  MoveL 2523 to (502.47, 492.57, 5) mm, rotated rx 0 ry 90 rz 0 deg; joints [-11.281, -26.8, 110.891, -15.281, -83.436, 50.783]
  Set speed (30.0 mm/s)
  Call Extruder(0.229)
  MoveL 2524 to (508.03, 498.13, 5) mm, rotated rx 0 ry 90 rz 0 deg; joints [-11.685, -26.677, 110.09, -15.709, -82.794, 51.008]
  MoveL 2525 to (508.16, 498.26, 5) mm, rotated rx 0 ry 90 rz 0 deg; joints [-11.694, -26.674, 110.072, -15.719, -82.78, 51.013]
  Set speed (120.0 mm/s)
  MoveL 2526 to (509.32, 490.68, 5) mm, rotated rx 0 ry 90 rz 0 deg; joints [-10.985, -26.681, 110.115, -15.004, -82.793, 50.925]
  Set speed (30.0 mm/s)
  Call Extruder(0.767)
  MoveL 2527 to (490.68, 509.32, 5) mm, rotated rx 0 ry 90 rz 0 deg; joints [-13.056, -26.94, 111.861, -17.04, -84.281, 50.715]
  MoveL 2528 to (490.56, 509.44, 5) mm, rotated rx 0 ry 90 rz 0 deg; joints [-13.07, -26.942, 111.873, -17.054, -84.29, 50.713]
  Set speed (120.0 mm/s)
  MoveL 2529 to (501.29, 492.36, 5) mm, rotated rx 0 ry 90 rz 0 deg; joints [-11.283, -26.822, 111.037, -15.28, -83.556, 50.75]
  Set speed (1000.0 mm/s)
  MoveL 2530 to (501.36, 492.29, 5) mm, rotated rx 0 ry 90 rz 0 deg; joints [-11.276, -26.821, 111.031, -15.272, -83.55, 50.751]
  Set speed (15.0 mm/s)
  Call Extruder(0.010)
  MoveL 2531 to (501.71, 492.29, 5) mm, rotated rx 0 ry 90 rz 0 deg; joints [-11.269, -26.815, 110.989, -15.267, -83.516, 50.76]
  Call Extruder(0.064)
  MoveL 2532 to (503.91, 492.29, 5) mm, rotated rx 0 ry 90 rz 0 deg; joints [-11.229, -26.775, 110.726, -15.233, -83.299, 50.815]
  Call Extruder(0.055)
  MoveL 2533 to (503.91, 490.4, 5) mm, rotated rx 0 ry 90 rz 0 deg; joints [-11.056, -26.782, 110.77, -15.057, -83.331, 50.787]
  Call Extruder(0.166)
  MoveL 2534 to (509.6, 490.4, 5) mm, rotated rx 0 ry 90 rz 0 deg; joints [-10.955, -26.677, 110.087, -14.974, -82.77, 50.927]
  Call Extruder(0.233)
  MoveL 2535 to (509.6, 498.42, 5) mm, rotated rx 0 ry 90 rz 0 deg; joints [-11.681, -26.646, 109.894, -15.711, -82.636, 51.053]
  Call Extruder(0.057)
  MoveL 2536 to (507.66, 498.42, 5) mm, rotated rx 0 ry 90 rz 0 deg; joints [-11.718, -26.683, 110.128, -15.741, -82.826, 51.003]
  Call Extruder(0.072)
  MoveL 2537 to (507.66, 500.9, 5) mm, rotated rx 0 ry 90 rz 0 deg; joints [-11.942, -26.673, 110.066, -15.969, -82.783, 51.042]
  Call Extruder(0.057)
  MoveL 2538 to (509.6, 500.9, 5) mm, rotated rx 0 ry 90 rz 0 deg; joints [-11.905, -26.636, 109.832, -15.939, -82.593, 51.093]
  Call Extruder(0.253)
  MoveL 2539 to (509.6, 509.6, 5) mm, rotated rx 0 ry 90 rz 0 deg; joints [-12.688, -26.599, 109.604, -16.735, -82.436, 51.238]
  Call Extruder(0.559)
  MoveL 2540 to (490.4, 509.6, 5) mm, rotated rx 0 ry 90 rz 0 deg; joints [-13.088, -26.944, 111.887, -17.072, -84.302, 50.711]
  MoveL 2541 to (490.4, 490.4, 5) mm, rotated rx 0 ry 90 rz 0 deg; joints [-11.303, -27.01, 112.375, -15.268, -84.666, 50.447]
  Call Extruder(0.144)
  MoveL 2542 to (495.34, 490.4, 5) mm, rotated rx 0 ry 90 rz 0 deg; joints [-11.211, -26.93, 111.791, -15.189, -84.177, 50.573]
  Call Extruder(0.055)
  MoveL 2543 to (495.35, 492.29, 5) mm, rotated rx 0 ry 90 rz 0 deg; joints [-11.387, -26.924, 111.746, -15.366, -84.144, 50.599]
  Call Extruder(0.072)
  MoveL 2544 to (497.81, 492.29, 5) mm, rotated rx 0 ry 90 rz 0 deg; joints [-11.341, -26.883, 111.454, -15.327, -83.901, 50.661]
  Call Extruder(0.055)
  MoveL 2545 to (497.81, 490.4, 5) mm, rotated rx 0 ry 90 rz 0 deg; joints [-11.166, -26.889, 111.499, -15.15, -83.934, 50.635]
  Call Extruder(0.093)
  MoveL 2546 to (501.01, 490.4, 5) mm, rotated rx 0 ry 90 rz 0 deg; joints [-11.108, -26.834, 111.117, -15.101, -83.617, 50.715]
  Call Extruder(0.010)
  MoveL 2547 to (501.36, 490.4, 5) mm, rotated rx 0 ry 90 rz 0 deg; joints [-11.102, -26.828, 111.075, -15.096, -83.583, 50.724]
  Call Extruder(0.007)
  MoveL 2548 to (501.36, 490.75, 5) mm, rotated rx 0 ry 90 rz 0 deg; joints [-11.134, -26.826, 111.067, -15.128, -83.577, 50.729]
  Call Extruder(0.035)
  MoveL 2549 to (501.36, 491.94, 5) mm, rotated rx 0 ry 90 rz 0 deg; joints [-11.244, -26.822, 111.039, -15.239, -83.556, 50.746]
  Call Extruder(0.007)
  MoveL 2550 to (501.36, 492.29, 5) mm, rotated rx 0 ry 90 rz 0 deg; joints [-11.276, -26.821, 111.031, -15.272, -83.55, 50.751]
  Set speed (120.0 mm/s)
  MoveL 2551 to (501.71, 492.29, 5) mm, rotated rx 0 ry 90 rz 0 deg; joints [-11.269, -26.815, 110.989, -15.267, -83.516, 50.76]
  Set speed (1000.0 mm/s)
  MoveL 2552 to (501.76, 492.29, 5) mm, rotated rx 0 ry 90 rz 0 deg; joints [-11.268, -26.814, 110.983, -15.266, -83.511, 50.761]
  Set speed (1000.0 mm/s)
  MoveL 2553 to (501.76, 492.99, 5) mm, rotated rx 0 ry 90 rz 0 deg; joints [-11.333, -26.811, 110.966, -15.331, -83.499, 50.771]
  Set speed (1000.0 mm/s)
  MoveL 2554 to (495.32, 492.32, 5) mm, rotated rx 0 ry 90 rz 0 deg; joints [-11.39, -26.924, 111.748, -15.369, -84.146, 50.598]
  Set speed (1000.0 mm/s)
  MoveL 2555 to (490.68, 490.68, 5) mm, rotated rx 0 ry 90 rz 0 deg; joints [-11.324, -27.005, 112.336, -15.29, -84.634, 50.458]
  Set speed (1000.0 mm/s)
  MoveL 2556 to (490.68, 490.68, 5.1) mm, rotated rx 0 ry 90 rz 0 deg; joints [-11.324, -27.015, 112.341, -15.29, -84.629, 50.459]
  Set speed (30.0 mm/s)
  Call Extruder(0.767)
  MoveL 2557 to (509.32, 509.32, 5.1) mm, rotated rx 0 ry 90 rz 0 deg; joints [-12.669, -26.616, 109.651, -16.714, -82.463, 51.227]
  MoveL 2558 to (509.44, 509.44, 5.1) mm, rotated rx 0 ry 90 rz 0 deg; joints [-12.677, -26.613, 109.632, -16.724, -82.449, 51.232]
  Set speed (120.0 mm/s)
  MoveL 2559 to (508.72, 501.17, 5.1) mm, rotated rx 0 ry 90 rz 0 deg; joints [-11.947, -26.662, 109.936, -15.978, -82.669, 51.076]
  Set speed (30.0 mm/s)
  Call Extruder(0.335)
  MoveL 2560 to (500.58, 509.32, 5.1) mm, rotated rx 0 ry 90 rz 0 deg; joints [-12.847, -26.781, 110.696, -16.863, -83.312, 50.99]
  Set speed (120.0 mm/s)
  MoveL 2561 to (499.42, 509.32, 5.1) mm, rotated rx 0 ry 90 rz 0 deg; joints [-12.872, -26.801, 110.833, -16.883, -83.425, 50.959]
  Set speed (30.0 mm/s)
  Call Extruder(0.360)
  MoveL 2562 to (490.68, 500.58, 5.1) mm, rotated rx 0 ry 90 rz 0 deg; joints [-12.247, -26.983, 112.098, -16.222, -84.447, 50.591]
  Set speed (120.0 mm/s)
  MoveL 2563 to (490.68, 499.42, 5.1) mm, rotated rx 0 ry 90 rz 0 deg; joints [-12.139, -26.987, 112.127, -16.113, -84.469, 50.575]
  Set speed (30.0 mm/s)
  Call Extruder(0.282)
  MoveL 2564 to (497.53, 492.57, 5.1) mm, rotated rx 0 ry 90 rz 0 deg; joints [-11.372, -26.897, 111.486, -15.358, -83.918, 50.659]
  Set speed (120.0 mm/s)
  MoveL 2565 to (498.14, 491.95, 5.1) mm, rotated rx 0 ry 90 rz 0 deg; joints [-11.304, -26.889, 111.427, -15.29, -83.868, 50.666]
  Set speed (30.0 mm/s)
  Call Extruder(0.052)
  MoveL 2566 to (499.42, 490.68, 5.1) mm, rotated rx 0 ry 90 rz 0 deg; joints [-11.163, -26.871, 111.305, -15.152, -83.764, 50.681]
  Set speed (120.0 mm/s)
  MoveL 2567 to (500.58, 490.68, 5.1) mm, rotated rx 0 ry 90 rz 0 deg; joints [-11.142, -26.851, 111.167, -15.134, -83.65, 50.71]
  Set speed (30.0 mm/s)
  Call Extruder(0.018)
  MoveL 2568 to (501.02, 491.12, 5.1) mm, rotated rx 0 ry 90 rz 0 deg; joints [-11.174, -26.842, 111.104, -15.168, -83.599, 50.727]
  Set speed (120.0 mm/s)
  MoveL 2569 to (502.47, 492.57, 5.1) mm, rotated rx 0 ry 90 rz 0 deg; joints [-11.281, -26.811, 110.897, -15.281, -83.431, 50.784]
  Set speed (30.0 mm/s)
  Call Extruder(0.229)
  MoveL 2570 to (508.03, 498.13, 5.1) mm, rotated rx 0 ry 90 rz 0 deg; joints [-11.685, -26.688, 110.095, -15.71, -82.789, 51.01]
  MoveL 2571 to (508.16, 498.26, 5.1) mm, rotated rx 0 ry 90 rz 0 deg; joints [-11.694, -26.685, 110.077, -15.719, -82.775, 51.015]
  Set speed (120.0 mm/s)
  MoveL 2572 to (509.32, 490.68, 5.1) mm, rotated rx 0 ry 90 rz 0 deg; joints [-10.985, -26.691, 110.12, -15.004, -82.788, 50.926]
  Set speed (30.0 mm/s)
  Call Extruder(0.767)
  MoveL 2573 to (490.68, 509.32, 5.1) mm, rotated rx 0 ry 90 rz 0 deg; joints [-13.056, -26.951, 111.867, -17.041, -84.276, 50.716]
  MoveL 2574 to (490.56, 509.44, 5.1) mm, rotated rx 0 ry 90 rz 0 deg; joints [-13.07, -26.952, 111.878, -17.054, -84.285, 50.715]
  Set speed (120.0 mm/s)
  MoveL 2575 to (507.59, 498.34, 5.1) mm, rotated rx 0 ry 90 rz 0 deg; joints [-11.712, -26.695, 110.143, -15.736, -82.829, 51.001]
  Set speed (1000.0 mm/s)
  MoveL 2576 to (507.66, 498.41, 5.1) mm, rotated rx 0 ry 90 rz 0 deg; joints [-11.717, -26.694, 110.133, -15.741, -82.821, 51.004]
  Set speed (15.0 mm/s)
  Call Extruder(0.072)
  MoveL 2577 to (507.66, 500.89, 5.1) mm, rotated rx 0 ry 90 rz 0 deg; joints [-11.942, -26.684, 110.071, -15.969, -82.778, 51.044]
  Call Extruder(0.057)
  MoveL 2578 to (509.6, 500.89, 5.1) mm, rotated rx 0 ry 90 rz 0 deg; joints [-11.905, -26.646, 109.837, -15.939, -82.588, 51.094]
  Call Extruder(0.253)
  MoveL 2579 to (509.6, 509.6, 5.1) mm, rotated rx 0 ry 90 rz 0 deg; joints [-12.688, -26.61, 109.609, -16.735, -82.431, 51.239]
  Call Extruder(0.559)
  MoveL 2580 to (490.4, 509.6, 5.1) mm, rotated rx 0 ry 90 rz 0 deg; joints [-13.088, -26.954, 111.892, -17.072, -84.297, 50.713]
  MoveL 2581 to (490.4, 490.4, 5.1) mm, rotated rx 0 ry 90 rz 0 deg; joints [-11.303, -27.021, 112.381, -15.268, -84.661, 50.449]
  Call Extruder(0.146)
  MoveL 2582 to (495.4, 490.4, 5.1) mm, rotated rx 0 ry 90 rz 0 deg; joints [-11.21, -26.94, 111.79, -15.188, -84.166, 50.576]
  Call Extruder(0.055)
  MoveL 2583 to (495.4, 492.29, 5.1) mm, rotated rx 0 ry 90 rz 0 deg; joints [-11.386, -26.934, 111.745, -15.366, -84.133, 50.601]
  Call Extruder(0.072)
  MoveL 2584 to (497.86, 492.29, 5.1) mm, rotated rx 0 ry 90 rz 0 deg; joints [-11.34, -26.892, 111.452, -15.326, -83.89, 50.664]
  Call Extruder(0.045)
  MoveL 2585 to (497.86, 490.75, 5.1) mm, rotated rx 0 ry 90 rz 0 deg; joints [-11.198, -26.897, 111.489, -15.182, -83.917, 50.643]
  Call Extruder(0.010)
  MoveL 2586 to (497.86, 490.4, 5.1) mm, rotated rx 0 ry 90 rz 0 deg; joints [-11.165, -26.899, 111.497, -15.15, -83.923, 50.638]
  Call Extruder(0.007)
  MoveL 2587 to (498.21, 490.4, 5.1) mm, rotated rx 0 ry 90 rz 0 deg; joints [-11.159, -26.893, 111.455, -15.144, -83.888, 50.647]
  Call Extruder(0.090)
  MoveL 2588 to (501.3, 490.4, 5.1) mm, rotated rx 0 ry 90 rz 0 deg; joints [-11.103, -26.839, 111.088, -15.097, -83.584, 50.724]
  Call Extruder(0.045)
  MoveL 2589 to (501.3, 491.94, 5.1) mm, rotated rx 0 ry 90 rz 0 deg; joints [-11.245, -26.834, 111.052, -15.24, -83.557, 50.746]
  Call Extruder(0.010)
  MoveL 2590 to (501.3, 492.29, 5.1) mm, rotated rx 0 ry 90 rz 0 deg; joints [-11.277, -26.833, 111.043, -15.273, -83.551, 50.751]
  Call Extruder(0.007)
  MoveL 2591 to (501.65, 492.29, 5.1) mm, rotated rx 0 ry 90 rz 0 deg; joints [-11.27, -26.826, 111.001, -15.268, -83.517, 50.76]
  Call Extruder(0.064)
  MoveL 2592 to (503.85, 492.29, 5.1) mm, rotated rx 0 ry 90 rz 0 deg; joints [-11.23, -26.787, 110.739, -15.234, -83.3, 50.815]
  Call Extruder(0.055)
  MoveL 2593 to (503.85, 490.41, 5.1) mm, rotated rx 0 ry 90 rz 0 deg; joints [-11.058, -26.794, 110.783, -15.059, -83.332, 50.787]
  Call Extruder(0.000)
  MoveL 2594 to (503.85, 490.4, 5.1) mm, rotated rx 0 ry 90 rz 0 deg; joints [-11.057, -26.794, 110.783, -15.058, -83.332, 50.787]
  Call Extruder(0.167)
  MoveL 2595 to (509.6, 490.4, 5.1) mm, rotated rx 0 ry 90 rz 0 deg; joints [-10.955, -26.687, 110.093, -14.974, -82.765, 50.929]
  Call Extruder(0.233)
  MoveL 2596 to (509.6, 498.41, 5.1) mm, rotated rx 0 ry 90 rz 0 deg; joints [-11.681, -26.656, 109.9, -15.711, -82.631, 51.054]
  Call Extruder(0.057)
  MoveL 2597 to (507.66, 498.41, 5.1) mm, rotated rx 0 ry 90 rz 0 deg; joints [-11.717, -26.694, 110.133, -15.741, -82.821, 51.004]
  Set speed (120.0 mm/s)
  MoveL 2598 to (507.66, 498.81, 5.1) mm, rotated rx 0 ry 90 rz 0 deg; joints [-11.754, -26.692, 110.123, -15.778, -82.814, 51.011]
  Set speed (1000.0 mm/s)
  MoveL 2599 to (506.96, 498.81, 5.1) mm, rotated rx 0 ry 90 rz 0 deg; joints [-11.767, -26.705, 110.207, -15.789, -82.883, 50.993]
  Set speed (1000.0 mm/s)
  MoveL 2600 to (490.68, 490.68, 5.1) mm, rotated rx 0 ry 90 rz 0 deg; joints [-11.324, -27.015, 112.341, -15.29, -84.629, 50.459]
  Set speed (1000.0 mm/s)
  MoveL 2601 to (490.68, 490.68, 5.2) mm, rotated rx 0 ry 90 rz 0 deg; joints [-11.324, -27.026, 112.347, -15.29, -84.623, 50.461]
  Set speed (30.0 mm/s)
  Call Extruder(0.767)
  MoveL 2602 to (509.32, 509.32, 5.2) mm, rotated rx 0 ry 90 rz 0 deg; joints [-12.669, -26.627, 109.656, -16.715, -82.458, 51.229]
  MoveL 2603 to (509.44, 509.44, 5.2) mm, rotated rx 0 ry 90 rz 0 deg; joints [-12.677, -26.624, 109.638, -16.724, -82.444, 51.234]
  Set speed (120.0 mm/s)
  MoveL 2604 to (508.72, 501.17, 5.2) mm, rotated rx 0 ry 90 rz 0 deg; joints [-11.947, -26.673, 109.941, -15.978, -82.664, 51.077]
  Set speed (30.0 mm/s)
  Call Extruder(0.335)
  MoveL 2605 to (500.58, 509.32, 5.2) mm, rotated rx 0 ry 90 rz 0 deg; joints [-12.847, -26.791, 110.701, -16.863, -83.307, 50.992]
  Set speed (120.0 mm/s)
  MoveL 2606 to (499.42, 509.32, 5.2) mm, rotated rx 0 ry 90 rz 0 deg; joints [-12.872, -26.812, 110.839, -16.883, -83.42, 50.96]
  Set speed (30.0 mm/s)
  Call Extruder(0.360)
  MoveL 2607 to (490.68, 500.58, 5.2) mm, rotated rx 0 ry 90 rz 0 deg; joints [-12.247, -26.993, 112.103, -16.222, -84.442, 50.593]
  Set speed (120.0 mm/s)
  MoveL 2608 to (490.68, 499.42, 5.2) mm, rotated rx 0 ry 90 rz 0 deg; joints [-12.139, -26.997, 112.133, -16.113, -84.463, 50.577]
  Set speed (30.0 mm/s)
  Call Extruder(0.282)
  MoveL 2609 to (497.53, 492.57, 5.2) mm, rotated rx 0 ry 90 rz 0 deg; joints [-11.372, -26.908, 111.491, -15.358, -83.913, 50.661]
  Set speed (120.0 mm/s)
  MoveL 2610 to (498.2, 491.9, 5.2) mm, rotated rx 0 ry 90 rz 0 deg; joints [-11.297, -26.898, 111.427, -15.284, -83.858, 50.668]
  Set speed (30.0 mm/s)
  Call Extruder(0.050)
  MoveL 2611 to (499.42, 490.68, 5.2) mm, rotated rx 0 ry 90 rz 0 deg; joints [-11.163, -26.882, 111.311, -15.152, -83.759, 50.682]
  Set speed (120.0 mm/s)
  MoveL 2612 to (500.58, 490.68, 5.2) mm, rotated rx 0 ry 90 rz 0 deg; joints [-11.141, -26.861, 111.173, -15.134, -83.645, 50.711]
  Set speed (30.0 mm/s)
  Call Extruder(0.016)
  MoveL 2613 to (500.96, 491.06, 5.2) mm, rotated rx 0 ry 90 rz 0 deg; joints [-11.169, -26.853, 111.118, -15.163, -83.601, 50.726]
  Set speed (120.0 mm/s)
  MoveL 2614 to (502.47, 492.57, 5.2) mm, rotated rx 0 ry 90 rz 0 deg; joints [-11.281, -26.821, 110.902, -15.281, -83.426, 50.786]
  Set speed (30.0 mm/s)
  Call Extruder(0.229)
  MoveL 2615 to (508.03, 498.13, 5.2) mm, rotated rx 0 ry 90 rz 0 deg; joints [-11.685, -26.698, 110.1, -15.71, -82.784, 51.011]
  MoveL 2616 to (508.15, 498.25, 5.2) mm, rotated rx 0 ry 90 rz 0 deg; joints [-11.694, -26.695, 110.083, -15.719, -82.77, 51.016]
  Set speed (120.0 mm/s)
  MoveL 2617 to (509.32, 490.68, 5.2) mm, rotated rx 0 ry 90 rz 0 deg; joints [-10.985, -26.702, 110.125, -15.004, -82.783, 50.927]
  Set speed (30.0 mm/s)
  Call Extruder(0.767)
  MoveL 2618 to (490.68, 509.32, 5.2) mm, rotated rx 0 ry 90 rz 0 deg; joints [-13.056, -26.961, 111.872, -17.041, -84.271, 50.718]
  MoveL 2619 to (490.56, 509.44, 5.2) mm, rotated rx 0 ry 90 rz 0 deg; joints [-13.07, -26.963, 111.883, -17.055, -84.28, 50.716]
  Set speed (120.0 mm/s)
  MoveL 2620 to (507.59, 498.34, 5.2) mm, rotated rx 0 ry 90 rz 0 deg; joints [-11.712, -26.706, 110.149, -15.736, -82.824, 51.003]
  Set speed (1000.0 mm/s)
  MoveL 2621 to (507.66, 498.41, 5.2) mm, rotated rx 0 ry 90 rz 0 deg; joints [-11.717, -26.704, 110.139, -15.741, -82.816, 51.006]
  Set speed (15.0 mm/s)
  Call Extruder(0.072)
  MoveL 2622 to (507.66, 500.89, 5.2) mm, rotated rx 0 ry 90 rz 0 deg; joints [-11.942, -26.694, 110.076, -15.969, -82.773, 51.045]
  Call Extruder(0.026)
  MoveL 2623 to (508.56, 500.9, 5.2) mm, rotated rx 0 ry 90 rz 0 deg; joints [-11.925, -26.677, 109.968, -15.955, -82.685, 51.069]
  Call Extruder(0.020)
  MoveL 2624 to (509.25, 500.89, 5.2) mm, rotated rx 0 ry 90 rz 0 deg; joints [-11.912, -26.664, 109.885, -15.944, -82.617, 51.086]
  Call Extruder(0.010)
  MoveL 2625 to (509.6, 500.89, 5.2) mm, rotated rx 0 ry 90 rz 0 deg; joints [-11.905, -26.657, 109.843, -15.939, -82.583, 51.095]
  Call Extruder(0.007)
  MoveL 2626 to (509.6, 501.24, 5.2) mm, rotated rx 0 ry 90 rz 0 deg; joints [-11.937, -26.656, 109.834, -15.971, -82.577, 51.101]
  Call Extruder(0.243)
  MoveL 2627 to (509.6, 509.6, 5.2) mm, rotated rx 0 ry 90 rz 0 deg; joints [-12.688, -26.62, 109.614, -16.736, -82.426, 51.241]
  Call Extruder(0.559)
  MoveL 2628 to (490.4, 509.6, 5.2) mm, rotated rx 0 ry 90 rz 0 deg; joints [-13.088, -26.965, 111.897, -17.072, -84.292, 50.714]
  MoveL 2629 to (490.4, 490.4, 5.2) mm, rotated rx 0 ry 90 rz 0 deg; joints [-11.303, -27.031, 112.386, -15.268, -84.656, 50.45]
  Call Extruder(0.147)
  MoveL 2630 to (495.46, 490.4, 5.2) mm, rotated rx 0 ry 90 rz 0 deg; joints [-11.209, -26.95, 111.788, -15.187, -84.156, 50.579]
  Call Extruder(0.055)
  MoveL 2631 to (495.46, 492.29, 5.2) mm, rotated rx 0 ry 90 rz 0 deg; joints [-11.385, -26.943, 111.743, -15.365, -84.122, 50.604]
  Call Extruder(0.062)
  MoveL 2632 to (497.57, 492.29, 5.2) mm, rotated rx 0 ry 90 rz 0 deg; joints [-11.345, -26.908, 111.492, -15.331, -83.914, 50.658]
  Call Extruder(0.010)
  MoveL 2633 to (497.92, 492.29, 5.2) mm, rotated rx 0 ry 90 rz 0 deg; joints [-11.339, -26.902, 111.45, -15.326, -83.879, 50.667]
  Call Extruder(0.007)
  MoveL 2634 to (497.92, 491.94, 5.2) mm, rotated rx 0 ry 90 rz 0 deg; joints [-11.307, -26.903, 111.459, -15.293, -83.885, 50.662]
  Call Extruder(0.045)
  MoveL 2635 to (497.92, 490.4, 5.2) mm, rotated rx 0 ry 90 rz 0 deg; joints [-11.164, -26.908, 111.495, -15.149, -83.912, 50.641]
  Call Extruder(0.097)
  MoveL 2636 to (501.24, 490.4, 5.2) mm, rotated rx 0 ry 90 rz 0 deg; joints [-11.104, -26.851, 111.1, -15.098, -83.584, 50.724]
  Call Extruder(0.045)
  MoveL 2637 to (501.24, 491.94, 5.2) mm, rotated rx 0 ry 90 rz 0 deg; joints [-11.246, -26.845, 111.064, -15.242, -83.558, 50.746]
  Call Extruder(0.010)
  MoveL 2638 to (501.24, 492.29, 5.2) mm, rotated rx 0 ry 90 rz 0 deg; joints [-11.278, -26.844, 111.056, -15.274, -83.552, 50.751]
  Call Extruder(0.007)
  MoveL 2639 to (501.59, 492.29, 5.2) mm, rotated rx 0 ry 90 rz 0 deg; joints [-11.272, -26.838, 111.014, -15.269, -83.518, 50.759]
  Call Extruder(0.064)
  MoveL 2640 to (503.79, 492.29, 5.2) mm, rotated rx 0 ry 90 rz 0 deg; joints [-11.231, -26.799, 110.751, -15.235, -83.301, 50.815]
  Call Extruder(0.054)
  MoveL 2641 to (503.79, 490.44, 5.2) mm, rotated rx 0 ry 90 rz 0 deg; joints [-11.062, -26.805, 110.795, -15.063, -83.332, 50.788]
  Call Extruder(0.001)
  MoveL 2642 to (503.79, 490.4, 5.2) mm, rotated rx 0 ry 90 rz 0 deg; joints [-11.058, -26.805, 110.796, -15.06, -83.333, 50.787]
  Call Extruder(0.169)
  MoveL 2643 to (509.6, 490.4, 5.2) mm, rotated rx 0 ry 90 rz 0 deg; joints [-10.955, -26.698, 110.098, -14.974, -82.76, 50.93]
  Call Extruder(0.233)
  MoveL 2644 to (509.6, 498.41, 5.2) mm, rotated rx 0 ry 90 rz 0 deg; joints [-11.681, -26.667, 109.905, -15.711, -82.626, 51.055]
  Call Extruder(0.057)
  MoveL 2645 to (507.66, 498.41, 5.2) mm, rotated rx 0 ry 90 rz 0 deg; joints [-11.717, -26.704, 110.139, -15.741, -82.816, 51.006]
  Set speed (120.0 mm/s)
  MoveL 2646 to (507.66, 498.81, 5.2) mm, rotated rx 0 ry 90 rz 0 deg; joints [-11.754, -26.702, 110.129, -15.778, -82.809, 51.012]
  Set speed (1000.0 mm/s)
  MoveL 2647 to (506.96, 498.81, 5.2) mm, rotated rx 0 ry 90 rz 0 deg; joints [-11.767, -26.716, 110.213, -15.789, -82.878, 50.994]
  Set speed (1000.0 mm/s)
  MoveL 2648 to (490.68, 490.68, 5.2) mm, rotated rx 0 ry 90 rz 0 deg; joints [-11.324, -27.026, 112.347, -15.29, -84.623, 50.461]
  Set speed (1000.0 mm/s)
  MoveL 2649 to (490.68, 490.68, 5.3) mm, rotated rx 0 ry 90 rz 0 deg; joints [-11.324, -27.037, 112.352, -15.29, -84.618, 50.462]
  Set speed (30.0 mm/s)
  Call Extruder(0.767)
  MoveL 2650 to (509.32, 509.32, 5.3) mm, rotated rx 0 ry 90 rz 0 deg; joints [-12.669, -26.637, 109.661, -16.715, -82.453, 51.23]
  MoveL 2651 to (509.44, 509.44, 5.3) mm, rotated rx 0 ry 90 rz 0 deg; joints [-12.677, -26.634, 109.643, -16.724, -82.439, 51.235]
  Set speed (120.0 mm/s)
  MoveL 2652 to (508.73, 501.17, 5.3) mm, rotated rx 0 ry 90 rz 0 deg; joints [-11.947, -26.683, 109.946, -15.978, -82.658, 51.079]
  Set speed (30.0 mm/s)
  Call Extruder(0.335)
  MoveL 2653 to (500.58, 509.32, 5.3) mm, rotated rx 0 ry 90 rz 0 deg; joints [-12.847, -26.802, 110.706, -16.863, -83.302, 50.993]
  Set speed (120.0 mm/s)
  MoveL 2654 to (499.42, 509.32, 5.3) mm, rotated rx 0 ry 90 rz 0 deg; joints [-12.872, -26.822, 110.844, -16.883, -83.415, 50.962]
  Set speed (30.0 mm/s)
  Call Extruder(0.360)
  MoveL 2655 to (490.68, 500.58, 5.3) mm, rotated rx 0 ry 90 rz 0 deg; joints [-12.247, -27.004, 112.109, -16.222, -84.436, 50.594]
  Set speed (120.0 mm/s)
  MoveL 2656 to (490.68, 499.42, 5.3) mm, rotated rx 0 ry 90 rz 0 deg; joints [-12.139, -27.008, 112.138, -16.113, -84.458, 50.578]
  Set speed (30.0 mm/s)
  Call Extruder(0.282)
  MoveL 2657 to (497.53, 492.57, 5.3) mm, rotated rx 0 ry 90 rz 0 deg; joints [-11.372, -26.918, 111.496, -15.358, -83.908, 50.662]
  Set speed (120.0 mm/s)
  MoveL 2658 to (498.26, 491.84, 5.3) mm, rotated rx 0 ry 90 rz 0 deg; joints [-11.291, -26.908, 111.426, -15.278, -83.849, 50.671]
  Set speed (30.0 mm/s)
  Call Extruder(0.048)
  MoveL 2659 to (499.42, 490.68, 5.3) mm, rotated rx 0 ry 90 rz 0 deg; joints [-11.163, -26.892, 111.316, -15.152, -83.754, 50.684]
  Set speed (120.0 mm/s)
  MoveL 2660 to (500.58, 490.68, 5.3) mm, rotated rx 0 ry 90 rz 0 deg; joints [-11.142, -26.872, 111.178, -15.134, -83.64, 50.713]
  Set speed (30.0 mm/s)
  Call Extruder(0.013)
  MoveL 2661 to (500.9, 491, 5.3) mm, rotated rx 0 ry 90 rz 0 deg; joints [-11.165, -26.865, 111.132, -15.159, -83.603, 50.725]
  Set speed (120.0 mm/s)
  MoveL 2662 to (502.47, 492.57, 5.3) mm, rotated rx 0 ry 90 rz 0 deg; joints [-11.281, -26.832, 110.907, -15.281, -83.421, 50.787]
  Set speed (30.0 mm/s)
  Call Extruder(0.229)
  MoveL 2663 to (508.03, 498.13, 5.3) mm, rotated rx 0 ry 90 rz 0 deg; joints [-11.685, -26.709, 110.106, -15.71, -82.78, 51.012]
  MoveL 2664 to (508.15, 498.25, 5.3) mm, rotated rx 0 ry 90 rz 0 deg; joints [-11.694, -26.706, 110.088, -15.719, -82.765, 51.017]
  Set speed (120.0 mm/s)
  MoveL 2665 to (509.32, 490.68, 5.3) mm, rotated rx 0 ry 90 rz 0 deg; joints [-10.985, -26.712, 110.131, -15.004, -82.778, 50.929]
  Set speed (30.0 mm/s)
  Call Extruder(0.767)
  MoveL 2666 to (490.68, 509.32, 5.3) mm, rotated rx 0 ry 90 rz 0 deg; joints [-13.056, -26.972, 111.877, -17.041, -84.266, 50.719]
  MoveL 2667 to (490.56, 509.44, 5.3) mm, rotated rx 0 ry 90 rz 0 deg; joints [-13.07, -26.974, 111.889, -17.055, -84.275, 50.718]
  Set speed (120.0 mm/s)
  MoveL 2668 to (507.59, 498.34, 5.3) mm, rotated rx 0 ry 90 rz 0 deg; joints [-11.712, -26.716, 110.154, -15.736, -82.819, 51.004]
  Set speed (1000.0 mm/s)
  MoveL 2669 to (507.66, 498.41, 5.3) mm, rotated rx 0 ry 90 rz 0 deg; joints [-11.717, -26.715, 110.144, -15.741, -82.811, 51.007]
  Set speed (15.0 mm/s)
  Call Extruder(0.072)
  MoveL 2670 to (507.66, 500.89, 5.3) mm, rotated rx 0 ry 90 rz 0 deg; joints [-11.942, -26.705, 110.081, -15.969, -82.768, 51.047]
  Call Extruder(0.057)
  MoveL 2671 to (509.6, 500.89, 5.3) mm, rotated rx 0 ry 90 rz 0 deg; joints [-11.905, -26.667, 109.848, -15.939, -82.578, 51.097]
  Call Extruder(0.253)
  MoveL 2672 to (509.6, 509.6, 5.3) mm, rotated rx 0 ry 90 rz 0 deg; joints [-12.688, -26.63, 109.62, -16.736, -82.421, 51.242]
  Call Extruder(0.559)
  MoveL 2673 to (490.4, 509.6, 5.3) mm, rotated rx 0 ry 90 rz 0 deg; joints [-13.088, -26.976, 111.903, -17.072, -84.287, 50.716]
  MoveL 2674 to (490.4, 490.4, 5.3) mm, rotated rx 0 ry 90 rz 0 deg; joints [-11.303, -27.042, 112.392, -15.268, -84.651, 50.452]
  Call Extruder(0.149)
  MoveL 2675 to (495.51, 490.4, 5.3) mm, rotated rx 0 ry 90 rz 0 deg; joints [-11.208, -26.959, 111.787, -15.187, -84.145, 50.581]
  Call Extruder(0.055)
  MoveL 2676 to (495.51, 492.29, 5.3) mm, rotated rx 0 ry 90 rz 0 deg; joints [-11.384, -26.953, 111.742, -15.364, -84.112, 50.607]
  Call Extruder(0.062)
  MoveL 2677 to (497.63, 492.29, 5.3) mm, rotated rx 0 ry 90 rz 0 deg; joints [-11.344, -26.917, 111.49, -15.33, -83.903, 50.661]
  Call Extruder(0.010)
  MoveL 2678 to (497.98, 492.29, 5.3) mm, rotated rx 0 ry 90 rz 0 deg; joints [-11.338, -26.911, 111.449, -15.325, -83.868, 50.67]
  Call Extruder(0.007)
  MoveL 2679 to (497.98, 491.94, 5.3) mm, rotated rx 0 ry 90 rz 0 deg; joints [-11.305, -26.913, 111.457, -15.292, -83.874, 50.665]
  Call Extruder(0.035)
  MoveL 2680 to (497.98, 490.75, 5.3) mm, rotated rx 0 ry 90 rz 0 deg; joints [-11.195, -26.917, 111.485, -15.181, -83.895, 50.648]
  Call Extruder(0.010)
  MoveL 2681 to (497.98, 490.4, 5.3) mm, rotated rx 0 ry 90 rz 0 deg; joints [-11.163, -26.918, 111.494, -15.148, -83.901, 50.644]
  Call Extruder(0.007)
  MoveL 2682 to (498.33, 490.4, 5.3) mm, rotated rx 0 ry 90 rz 0 deg; joints [-11.157, -26.912, 111.452, -15.143, -83.866, 50.652]
  Call Extruder(0.073)
  MoveL 2683 to (500.83, 490.4, 5.3) mm, rotated rx 0 ry 90 rz 0 deg; joints [-11.111, -26.869, 111.155, -15.104, -83.62, 50.715]
  Call Extruder(0.010)
  MoveL 2684 to (501.18, 490.4, 5.3) mm, rotated rx 0 ry 90 rz 0 deg; joints [-11.105, -26.862, 111.113, -15.099, -83.585, 50.724]
  Call Extruder(0.007)
  MoveL 2685 to (501.18, 490.75, 5.3) mm, rotated rx 0 ry 90 rz 0 deg; joints [-11.137, -26.861, 111.105, -15.132, -83.579, 50.728]
  Call Extruder(0.035)
  MoveL 2686 to (501.18, 491.94, 5.3) mm, rotated rx 0 ry 90 rz 0 deg; joints [-11.247, -26.857, 111.077, -15.243, -83.559, 50.745]
  Call Extruder(0.010)
  MoveL 2687 to (501.18, 492.29, 5.3) mm, rotated rx 0 ry 90 rz 0 deg; joints [-11.279, -26.856, 111.068, -15.275, -83.553, 50.751]
  Call Extruder(0.007)
  MoveL 2688 to (501.53, 492.29, 5.3) mm, rotated rx 0 ry 90 rz 0 deg; joints [-11.273, -26.85, 111.027, -15.27, -83.519, 50.759]
  Call Extruder(0.064)
  MoveL 2689 to (503.72, 492.29, 5.3) mm, rotated rx 0 ry 90 rz 0 deg; joints [-11.233, -26.81, 110.764, -15.236, -83.303, 50.814]
  Call Extruder(0.055)
  MoveL 2690 to (503.72, 490.4, 5.3) mm, rotated rx 0 ry 90 rz 0 deg; joints [-11.059, -26.817, 110.809, -15.061, -83.334, 50.787]
  Call Extruder(0.171)
  MoveL 2691 to (509.6, 490.4, 5.3) mm, rotated rx 0 ry 90 rz 0 deg; joints [-10.955, -26.708, 110.103, -14.974, -82.755, 50.931]
  Call Extruder(0.233)
  MoveL 2692 to (509.6, 498.41, 5.3) mm, rotated rx 0 ry 90 rz 0 deg; joints [-11.681, -26.677, 109.91, -15.711, -82.621, 51.057]
  Call Extruder(0.057)
  MoveL 2693 to (507.66, 498.41, 5.3) mm, rotated rx 0 ry 90 rz 0 deg; joints [-11.717, -26.715, 110.144, -15.741, -82.811, 51.007]
  Set speed (120.0 mm/s)
  MoveL 2694 to (507.66, 498.81, 5.3) mm, rotated rx 0 ry 90 rz 0 deg; joints [-11.754, -26.713, 110.134, -15.778, -82.804, 51.014]
  Set speed (1000.0 mm/s)
  MoveL 2695 to (506.96, 498.81, 5.3) mm, rotated rx 0 ry 90 rz 0 deg; joints [-11.767, -26.726, 110.218, -15.789, -82.873, 50.996]
  Set speed (1000.0 mm/s)
  MoveL 2696 to (490.68, 490.68, 5.3) mm, rotated rx 0 ry 90 rz 0 deg; joints [-11.324, -27.037, 112.352, -15.29, -84.618, 50.462]
  Set speed (1000.0 mm/s)
  MoveL 2697 to (490.68, 490.68, 5.4) mm, rotated rx 0 ry 90 rz 0 deg; joints [-11.324, -27.047, 112.357, -15.29, -84.613, 50.464]
  Set speed (30.0 mm/s)
  Call Extruder(0.767)
  MoveL 2698 to (509.32, 509.32, 5.4) mm, rotated rx 0 ry 90 rz 0 deg; joints [-12.669, -26.648, 109.666, -16.715, -82.449, 51.232]
  MoveL 2699 to (509.44, 509.44, 5.4) mm, rotated rx 0 ry 90 rz 0 deg; joints [-12.677, -26.645, 109.648, -16.724, -82.434, 51.237]
  Set speed (120.0 mm/s)
  MoveL 2700 to (508.73, 501.17, 5.4) mm, rotated rx 0 ry 90 rz 0 deg; joints [-11.947, -26.694, 109.951, -15.978, -82.653, 51.08]
  Set speed (30.0 mm/s)
  Call Extruder(0.335)
  MoveL 2701 to (500.58, 509.32, 5.4) mm, rotated rx 0 ry 90 rz 0 deg; joints [-12.847, -26.812, 110.711, -16.863, -83.297, 50.995]
  Set speed (120.0 mm/s)
  MoveL 2702 to (499.42, 509.32, 5.4) mm, rotated rx 0 ry 90 rz 0 deg; joints [-12.872, -26.833, 110.849, -16.883, -83.41, 50.963]
  Set speed (30.0 mm/s)
  Call Extruder(0.360)
  MoveL 2703 to (490.68, 500.58, 5.4) mm, rotated rx 0 ry 90 rz 0 deg; joints [-12.247, -27.014, 112.114, -16.222, -84.431, 50.596]
  Set speed (120.0 mm/s)
  MoveL 2704 to (490.68, 499.42, 5.4) mm, rotated rx 0 ry 90 rz 0 deg; joints [-12.139, -27.018, 112.143, -16.114, -84.453, 50.58]
  Set speed (30.0 mm/s)
  Call Extruder(0.282)
  MoveL 2705 to (497.53, 492.57, 5.4) mm, rotated rx 0 ry 90 rz 0 deg; joints [-11.372, -26.929, 111.502, -15.358, -83.903, 50.664]
  Set speed (120.0 mm/s)
  MoveL 2706 to (498.32, 491.78, 5.4) mm, rotated rx 0 ry 90 rz 0 deg; joints [-11.284, -26.918, 111.426, -15.272, -83.839, 50.673]
  Set speed (30.0 mm/s)
  Call Extruder(0.045)
  MoveL 2707 to (499.42, 490.68, 5.4) mm, rotated rx 0 ry 90 rz 0 deg; joints [-11.163, -26.903, 111.321, -15.152, -83.749, 50.685]
  Set speed (120.0 mm/s)
  MoveL 2708 to (500.58, 490.68, 5.4) mm, rotated rx 0 ry 90 rz 0 deg; joints [-11.142, -26.883, 111.183, -15.134, -83.635, 50.714]
  Set speed (30.0 mm/s)
  Call Extruder(0.011)
  MoveL 2709 to (500.84, 490.94, 5.4) mm, rotated rx 0 ry 90 rz 0 deg; joints [-11.161, -26.877, 111.146, -15.154, -83.605, 50.724]
  Set speed (120.0 mm/s)
  MoveL 2710 to (501.09, 492.32, 5.4) mm, rotated rx 0 ry 90 rz 0 deg; joints [-11.283, -26.868, 111.084, -15.279, -83.557, 50.75]
  Set speed (1000.0 mm/s)
  MoveL 2711 to (502.47, 492.57, 5.4) mm, rotated rx 0 ry 90 rz 0 deg; joints [-11.281, -26.842, 110.912, -15.282, -83.416, 50.789]
  Set speed (30.0 mm/s)
  Call Extruder(0.229)
  MoveL 2712 to (508.03, 498.13, 5.4) mm, rotated rx 0 ry 90 rz 0 deg; joints [-11.685, -26.719, 110.111, -15.71, -82.775, 51.014]
  MoveL 2713 to (508.15, 498.25, 5.4) mm, rotated rx 0 ry 90 rz 0 deg; joints [-11.694, -26.716, 110.093, -15.719, -82.76, 51.019]
  Set speed (120.0 mm/s)
  MoveL 2714 to (509.32, 490.68, 5.4) mm, rotated rx 0 ry 90 rz 0 deg; joints [-10.985, -26.723, 110.136, -15.004, -82.773, 50.93]
  Set speed (30.0 mm/s)
  Call Extruder(0.767)
  MoveL 2715 to (490.68, 509.32, 5.4) mm, rotated rx 0 ry 90 rz 0 deg; joints [-13.056, -26.983, 111.883, -17.041, -84.261, 50.721]
  MoveL 2716 to (490.56, 509.44, 5.4) mm, rotated rx 0 ry 90 rz 0 deg; joints [-13.07, -26.984, 111.894, -17.055, -84.27, 50.719]
  Set speed (120.0 mm/s)
  MoveL 2717 to (507.59, 498.34, 5.4) mm, rotated rx 0 ry 90 rz 0 deg; joints [-11.712, -26.727, 110.159, -15.736, -82.814, 51.006]
  Set speed (1000.0 mm/s)
  MoveL 2718 to (507.66, 498.41, 5.4) mm, rotated rx 0 ry 90 rz 0 deg; joints [-11.717, -26.725, 110.149, -15.741, -82.806, 51.009]
  Set speed (15.0 mm/s)
  Call Extruder(0.072)
  MoveL 2719 to (507.66, 500.89, 5.4) mm, rotated rx 0 ry 90 rz 0 deg; joints [-11.942, -26.715, 110.087, -15.969, -82.763, 51.048]
  Call Extruder(0.057)
  MoveL 2720 to (509.6, 500.89, 5.4) mm, rotated rx 0 ry 90 rz 0 deg; joints [-11.905, -26.678, 109.853, -15.939, -82.573, 51.098]
  Call Extruder(0.253)
  MoveL 2721 to (509.6, 509.6, 5.4) mm, rotated rx 0 ry 90 rz 0 deg; joints [-12.688, -26.641, 109.625, -16.736, -82.416, 51.244]
  Call Extruder(0.559)
  MoveL 2722 to (490.4, 509.6, 5.4) mm, rotated rx 0 ry 90 rz 0 deg; joints [-13.088, -26.986, 111.908, -17.072, -84.282, 50.717]
  MoveL 2723 to (490.4, 490.4, 5.4) mm, rotated rx 0 ry 90 rz 0 deg; joints [-11.303, -27.053, 112.397, -15.269, -84.646, 50.453]
  Call Extruder(0.150)
  MoveL 2724 to (495.57, 490.4, 5.4) mm, rotated rx 0 ry 90 rz 0 deg; joints [-11.207, -26.969, 111.786, -15.186, -84.135, 50.584]
  Call Extruder(0.045)
  MoveL 2725 to (495.57, 491.94, 5.4) mm, rotated rx 0 ry 90 rz 0 deg; joints [-11.35, -26.964, 111.749, -15.331, -84.107, 50.605]
  Call Extruder(0.010)
  MoveL 2726 to (495.57, 492.29, 5.4) mm, rotated rx 0 ry 90 rz 0 deg; joints [-11.383, -26.963, 111.741, -15.363, -84.101, 50.61]
  Call Extruder(0.007)
  MoveL 2727 to (495.92, 492.29, 5.4) mm, rotated rx 0 ry 90 rz 0 deg; joints [-11.376, -26.957, 111.699, -15.358, -84.067, 50.619]
  Call Extruder(0.062)
  MoveL 2728 to (498.04, 492.29, 5.4) mm, rotated rx 0 ry 90 rz 0 deg; joints [-11.337, -26.921, 111.447, -15.324, -83.857, 50.673]
  Call Extruder(0.045)
  MoveL 2729 to (498.04, 490.75, 5.4) mm, rotated rx 0 ry 90 rz 0 deg; joints [-11.194, -26.926, 111.484, -15.18, -83.884, 50.651]
  Call Extruder(0.010)
  MoveL 2730 to (498.04, 490.4, 5.4) mm, rotated rx 0 ry 90 rz 0 deg; joints [-11.162, -26.927, 111.492, -15.147, -83.89, 50.646]
  Call Extruder(0.007)
  MoveL 2731 to (498.39, 490.4, 5.4) mm, rotated rx 0 ry 90 rz 0 deg; joints [-11.156, -26.921, 111.45, -15.142, -83.855, 50.655]
  Call Extruder(0.079)
  MoveL 2732 to (501.12, 490.4, 5.4) mm, rotated rx 0 ry 90 rz 0 deg; joints [-11.106, -26.874, 111.126, -15.1, -83.586, 50.723]
  Call Extruder(0.045)
  MoveL 2733 to (501.12, 491.94, 5.4) mm, rotated rx 0 ry 90 rz 0 deg; joints [-11.248, -26.869, 111.089, -15.244, -83.56, 50.745]
  Call Extruder(0.010)
  MoveL 2734 to (501.12, 492.29, 5.4) mm, rotated rx 0 ry 90 rz 0 deg; joints [-11.28, -26.868, 111.081, -15.276, -83.554, 50.75]
  Call Extruder(0.007)
  MoveL 2735 to (501.47, 492.29, 5.4) mm, rotated rx 0 ry 90 rz 0 deg; joints [-11.274, -26.861, 111.039, -15.271, -83.52, 50.759]
  Call Extruder(0.064)
  MoveL 2736 to (503.66, 492.29, 5.4) mm, rotated rx 0 ry 90 rz 0 deg; joints [-11.234, -26.822, 110.777, -15.238, -83.304, 50.814]
  Call Extruder(0.055)
  MoveL 2737 to (503.66, 490.4, 5.4) mm, rotated rx 0 ry 90 rz 0 deg; joints [-11.06, -26.829, 110.822, -15.062, -83.335, 50.787]
  Call Extruder(0.173)
  MoveL 2738 to (509.6, 490.4, 5.4) mm, rotated rx 0 ry 90 rz 0 deg; joints [-10.955, -26.719, 110.109, -14.975, -82.75, 50.933]
  Call Extruder(0.233)
  MoveL 2739 to (509.6, 498.41, 5.4) mm, rotated rx 0 ry 90 rz 0 deg; joints [-11.681, -26.688, 109.916, -15.712, -82.616, 51.058]
  Call Extruder(0.057)
  MoveL 2740 to (507.66, 498.41, 5.4) mm, rotated rx 0 ry 90 rz 0 deg; joints [-11.717, -26.725, 110.149, -15.741, -82.806, 51.009]
  Set speed (120.0 mm/s)
  MoveL 2741 to (507.66, 498.81, 5.4) mm, rotated rx 0 ry 90 rz 0 deg; joints [-11.753, -26.723, 110.139, -15.778, -82.799, 51.015]
  Set speed (1000.0 mm/s)
  MoveL 2742 to (506.96, 498.81, 5.4) mm, rotated rx 0 ry 90 rz 0 deg; joints [-11.767, -26.737, 110.223, -15.789, -82.868, 50.997]
  Set speed (1000.0 mm/s)
  MoveL 2743 to (490.68, 490.68, 5.4) mm, rotated rx 0 ry 90 rz 0 deg; joints [-11.324, -27.047, 112.357, -15.29, -84.613, 50.464]
  Set speed (1000.0 mm/s)
  MoveL 2744 to (490.68, 490.68, 5.5) mm, rotated rx 0 ry 90 rz 0 deg; joints [-11.324, -27.058, 112.363, -15.29, -84.608, 50.465]
  Set speed (30.0 mm/s)
  Call Extruder(0.767)
  MoveL 2745 to (509.32, 509.32, 5.5) mm, rotated rx 0 ry 90 rz 0 deg; joints [-12.669, -26.658, 109.672, -16.715, -82.444, 51.233]
  MoveL 2746 to (509.44, 509.44, 5.5) mm, rotated rx 0 ry 90 rz 0 deg; joints [-12.677, -26.655, 109.654, -16.724, -82.429, 51.238]
  Set speed (120.0 mm/s)
  MoveL 2747 to (508.73, 501.17, 5.5) mm, rotated rx 0 ry 90 rz 0 deg; joints [-11.947, -26.704, 109.956, -15.979, -82.648, 51.082]
  Set speed (30.0 mm/s)
  Call Extruder(0.335)
  MoveL 2748 to (500.58, 509.32, 5.5) mm, rotated rx 0 ry 90 rz 0 deg; joints [-12.847, -26.823, 110.717, -16.863, -83.292, 50.996]
  Set speed (120.0 mm/s)
  MoveL 2749 to (499.42, 509.32, 5.5) mm, rotated rx 0 ry 90 rz 0 deg; joints [-12.872, -26.843, 110.855, -16.884, -83.405, 50.965]
  Set speed (30.0 mm/s)
  Call Extruder(0.360)
  MoveL 2750 to (490.68, 500.58, 5.5) mm, rotated rx 0 ry 90 rz 0 deg; joints [-12.247, -27.025, 112.119, -16.223, -84.426, 50.597]
  Set speed (120.0 mm/s)
  MoveL 2751 to (490.68, 499.42, 5.5) mm, rotated rx 0 ry 90 rz 0 deg; joints [-12.139, -27.029, 112.149, -16.114, -84.448, 50.581]
  Set speed (30.0 mm/s)
  Call Extruder(0.282)
  MoveL 2752 to (497.53, 492.57, 5.5) mm, rotated rx 0 ry 90 rz 0 deg; joints [-11.372, -26.939, 111.507, -15.358, -83.898, 50.665]
  Set speed (120.0 mm/s)
  MoveL 2753 to (498.38, 491.72, 5.5) mm, rotated rx 0 ry 90 rz 0 deg; joints [-11.277, -26.928, 111.426, -15.265, -83.829, 50.675]
  Set speed (30.0 mm/s)
  Call Extruder(0.043)
  MoveL 2754 to (499.42, 490.68, 5.5) mm, rotated rx 0 ry 90 rz 0 deg; joints [-11.163, -26.913, 111.327, -15.152, -83.744, 50.686]
  Set speed (120.0 mm/s)
  MoveL 2755 to (500.58, 490.68, 5.5) mm, rotated rx 0 ry 90 rz 0 deg; joints [-11.142, -26.893, 111.188, -15.134, -83.63, 50.715]
  Set speed (30.0 mm/s)
  Call Extruder(0.008)
  MoveL 2756 to (500.78, 490.88, 5.5) mm, rotated rx 0 ry 90 rz 0 deg; joints [-11.156, -26.889, 111.16, -15.15, -83.607, 50.723]
  Set speed (120.0 mm/s)
  MoveL 2757 to (501.03, 492.32, 5.5) mm, rotated rx 0 ry 90 rz 0 deg; joints [-11.284, -26.88, 111.096, -15.28, -83.558, 50.75]
  Set speed (1000.0 mm/s)
  MoveL 2758 to (502.47, 492.57, 5.5) mm, rotated rx 0 ry 90 rz 0 deg; joints [-11.281, -26.853, 110.918, -15.282, -83.411, 50.79]
  Set speed (30.0 mm/s)
  Call Extruder(0.229)
  MoveL 2759 to (508.03, 498.13, 5.5) mm, rotated rx 0 ry 90 rz 0 deg; joints [-11.685, -26.73, 110.117, -15.71, -82.77, 51.015]
  MoveL 2760 to (508.15, 498.25, 5.5) mm, rotated rx 0 ry 90 rz 0 deg; joints [-11.693, -26.727, 110.099, -15.719, -82.756, 51.02]
  Set speed (120.0 mm/s)
  MoveL 2761 to (509.32, 490.68, 5.5) mm, rotated rx 0 ry 90 rz 0 deg; joints [-10.985, -26.733, 110.141, -15.005, -82.768, 50.931]
  Set speed (30.0 mm/s)
  Call Extruder(0.767)
  MoveL 2762 to (490.68, 509.32, 5.5) mm, rotated rx 0 ry 90 rz 0 deg; joints [-13.056, -26.993, 111.888, -17.041, -84.256, 50.722]
  MoveL 2763 to (490.56, 509.44, 5.5) mm, rotated rx 0 ry 90 rz 0 deg; joints [-13.07, -26.995, 111.899, -17.055, -84.265, 50.721]
  Set speed (120.0 mm/s)
  MoveL 2764 to (507.59, 498.34, 5.5) mm, rotated rx 0 ry 90 rz 0 deg; joints [-11.712, -26.737, 110.164, -15.736, -82.809, 51.007]
  Set speed (1000.0 mm/s)
  MoveL 2765 to (507.66, 498.41, 5.5) mm, rotated rx 0 ry 90 rz 0 deg; joints [-11.717, -26.735, 110.154, -15.742, -82.801, 51.01]
  Set speed (15.0 mm/s)
  Call Extruder(0.072)
  MoveL 2766 to (507.66, 500.89, 5.5) mm, rotated rx 0 ry 90 rz 0 deg; joints [-11.942, -26.726, 110.092, -15.97, -82.758, 51.05]
  Call Extruder(0.057)
  MoveL 2767 to (509.6, 500.89, 5.5) mm, rotated rx 0 ry 90 rz 0 deg; joints [-11.905, -26.688, 109.859, -15.939, -82.568, 51.1]
  Call Extruder(0.253)
  MoveL 2768 to (509.6, 509.6, 5.5) mm, rotated rx 0 ry 90 rz 0 deg; joints [-12.688, -26.651, 109.63, -16.736, -82.411, 51.245]
  Call Extruder(0.559)
  MoveL 2769 to (490.4, 509.6, 5.5) mm, rotated rx 0 ry 90 rz 0 deg; joints [-13.088, -26.997, 111.913, -17.073, -84.277, 50.719]
  MoveL 2770 to (490.4, 490.4, 5.5) mm, rotated rx 0 ry 90 rz 0 deg; joints [-11.303, -27.063, 112.402, -15.269, -84.641, 50.454]
  Call Extruder(0.152)
  MoveL 2771 to (495.62, 490.4, 5.5) mm, rotated rx 0 ry 90 rz 0 deg; joints [-11.206, -26.979, 111.785, -15.185, -84.124, 50.587]
  Call Extruder(0.055)
  MoveL 2772 to (495.62, 492.29, 5.5) mm, rotated rx 0 ry 90 rz 0 deg; joints [-11.382, -26.972, 111.739, -15.363, -84.091, 50.613]
  Call Extruder(0.072)
  MoveL 2773 to (498.1, 492.29, 5.5) mm, rotated rx 0 ry 90 rz 0 deg; joints [-11.336, -26.931, 111.445, -15.323, -83.846, 50.676]
  Call Extruder(0.045)
  MoveL 2774 to (498.1, 490.75, 5.5) mm, rotated rx 0 ry 90 rz 0 deg; joints [-11.193, -26.936, 111.482, -15.179, -83.873, 50.654]
  Call Extruder(0.010)
  MoveL 2775 to (498.1, 490.4, 5.5) mm, rotated rx 0 ry 90 rz 0 deg; joints [-11.161, -26.937, 111.49, -15.146, -83.879, 50.649]
  Call Extruder(0.007)
  MoveL 2776 to (498.45, 490.4, 5.5) mm, rotated rx 0 ry 90 rz 0 deg; joints [-11.154, -26.931, 111.448, -15.141, -83.844, 50.658]
  Call Extruder(0.076)
  MoveL 2777 to (501.06, 490.4, 5.5) mm, rotated rx 0 ry 90 rz 0 deg; joints [-11.107, -26.886, 111.138, -15.101, -83.587, 50.723]
  Call Extruder(0.045)
  MoveL 2778 to (501.06, 491.94, 5.5) mm, rotated rx 0 ry 90 rz 0 deg; joints [-11.249, -26.88, 111.102, -15.245, -83.561, 50.745]
  Call Extruder(0.010)
  MoveL 2779 to (501.05, 492.29, 5.5) mm, rotated rx 0 ry 90 rz 0 deg; joints [-11.281, -26.879, 111.094, -15.277, -83.555, 50.75]
  Call Extruder(0.007)
  MoveL 2780 to (501.4, 492.29, 5.5) mm, rotated rx 0 ry 90 rz 0 deg; joints [-11.275, -26.873, 111.052, -15.272, -83.521, 50.759]
  Call Extruder(0.064)
  MoveL 2781 to (503.6, 492.29, 5.5) mm, rotated rx 0 ry 90 rz 0 deg; joints [-11.235, -26.834, 110.79, -15.239, -83.305, 50.814]
  Call Extruder(0.055)
  MoveL 2782 to (503.6, 490.4, 5.5) mm, rotated rx 0 ry 90 rz 0 deg; joints [-11.061, -26.84, 110.834, -15.063, -83.337, 50.786]
  Call Extruder(0.175)
  MoveL 2783 to (509.6, 490.4, 5.5) mm, rotated rx 0 ry 90 rz 0 deg; joints [-10.955, -26.729, 110.114, -14.975, -82.745, 50.934]
  Call Extruder(0.233)
  MoveL 2784 to (509.6, 498.41, 5.5) mm, rotated rx 0 ry 90 rz 0 deg; joints [-11.681, -26.698, 109.921, -15.712, -82.611, 51.06]
  Call Extruder(0.057)
  MoveL 2785 to (507.66, 498.41, 5.5) mm, rotated rx 0 ry 90 rz 0 deg; joints [-11.717, -26.735, 110.154, -15.742, -82.801, 51.01]
  Set speed (120.0 mm/s)
  MoveL 2786 to (507.66, 498.81, 5.5) mm, rotated rx 0 ry 90 rz 0 deg; joints [-11.753, -26.734, 110.144, -15.778, -82.794, 51.016]
  Set speed (1000.0 mm/s)
  MoveL 2787 to (506.96, 498.81, 5.5) mm, rotated rx 0 ry 90 rz 0 deg; joints [-11.767, -26.747, 110.228, -15.789, -82.863, 50.998]
  Set speed (1000.0 mm/s)
  MoveL 2788 to (490.68, 490.68, 5.5) mm, rotated rx 0 ry 90 rz 0 deg; joints [-11.324, -27.058, 112.363, -15.29, -84.608, 50.465]
  Set speed (1000.0 mm/s)
  MoveL 2789 to (490.68, 490.68, 5.6) mm, rotated rx 0 ry 90 rz 0 deg; joints [-11.324, -27.069, 112.368, -15.291, -84.603, 50.466]
  Set speed (30.0 mm/s)
  Call Extruder(0.767)
  MoveL 2790 to (509.32, 509.32, 5.6) mm, rotated rx 0 ry 90 rz 0 deg; joints [-12.669, -26.668, 109.677, -16.715, -82.439, 51.235]
  MoveL 2791 to (509.44, 509.44, 5.6) mm, rotated rx 0 ry 90 rz 0 deg; joints [-12.677, -26.666, 109.659, -16.724, -82.424, 51.24]
  Set speed (120.0 mm/s)
  MoveL 2792 to (508.73, 501.17, 5.6) mm, rotated rx 0 ry 90 rz 0 deg; joints [-11.946, -26.714, 109.962, -15.979, -82.643, 51.083]
  Set speed (30.0 mm/s)
  Call Extruder(0.335)
  MoveL 2793 to (500.58, 509.32, 5.6) mm, rotated rx 0 ry 90 rz 0 deg; joints [-12.847, -26.833, 110.722, -16.864, -83.287, 50.998]
  Set speed (120.0 mm/s)
  MoveL 2794 to (499.42, 509.32, 5.6) mm, rotated rx 0 ry 90 rz 0 deg; joints [-12.872, -26.854, 110.86, -16.884, -83.4, 50.966]
  Set speed (30.0 mm/s)
  Call Extruder(0.360)
  MoveL 2795 to (490.68, 500.58, 5.6) mm, rotated rx 0 ry 90 rz 0 deg; joints [-12.247, -27.036, 112.125, -16.223, -84.421, 50.599]
  Set speed (120.0 mm/s)
  MoveL 2796 to (490.68, 499.42, 5.6) mm, rotated rx 0 ry 90 rz 0 deg; joints [-12.139, -27.04, 112.154, -16.114, -84.443, 50.583]
  Set speed (30.0 mm/s)
  Call Extruder(0.282)
  MoveL 2797 to (497.53, 492.57, 5.6) mm, rotated rx 0 ry 90 rz 0 deg; joints [-11.372, -26.95, 111.512, -15.359, -83.893, 50.666]
  Set speed (120.0 mm/s)
  MoveL 2798 to (498.44, 491.66, 5.6) mm, rotated rx 0 ry 90 rz 0 deg; joints [-11.271, -26.937, 111.425, -15.259, -83.819, 50.677]
  Set speed (30.0 mm/s)
  Call Extruder(0.040)
  MoveL 2799 to (499.42, 490.68, 5.6) mm, rotated rx 0 ry 90 rz 0 deg; joints [-11.163, -26.924, 111.332, -15.152, -83.739, 50.688]
  Set speed (120.0 mm/s)
  MoveL 2800 to (500.58, 490.68, 5.6) mm, rotated rx 0 ry 90 rz 0 deg; joints [-11.142, -26.904, 111.194, -15.135, -83.625, 50.717]
  Set speed (30.0 mm/s)
  Call Extruder(0.006)
  MoveL 2801 to (500.71, 490.81, 5.6) mm, rotated rx 0 ry 90 rz 0 deg; joints [-11.151, -26.901, 111.174, -15.145, -83.609, 50.722]
  Set speed (120.0 mm/s)
  MoveL 2802 to (500.97, 492.32, 5.6) mm, rotated rx 0 ry 90 rz 0 deg; joints [-11.286, -26.891, 111.109, -15.282, -83.558, 50.75]
  Set speed (1000.0 mm/s)
  MoveL 2803 to (502.47, 492.57, 5.6) mm, rotated rx 0 ry 90 rz 0 deg; joints [-11.281, -26.863, 110.923, -15.282, -83.406, 50.791]
  Set speed (30.0 mm/s)
  Call Extruder(0.229)
  MoveL 2804 to (508.03, 498.13, 5.6) mm, rotated rx 0 ry 90 rz 0 deg; joints [-11.685, -26.74, 110.122, -15.71, -82.765, 51.016]
  MoveL 2805 to (508.15, 498.25, 5.6) mm, rotated rx 0 ry 90 rz 0 deg; joints [-11.693, -26.737, 110.104, -15.719, -82.751, 51.021]
  Set speed (120.0 mm/s)
  MoveL 2806 to (509.32, 490.68, 5.6) mm, rotated rx 0 ry 90 rz 0 deg; joints [-10.985, -26.744, 110.146, -15.005, -82.763, 50.933]
  Set speed (30.0 mm/s)
  Call Extruder(0.767)
  MoveL 2807 to (490.68, 509.32, 5.6) mm, rotated rx 0 ry 90 rz 0 deg; joints [-13.056, -27.004, 111.893, -17.041, -84.251, 50.724]
  MoveL 2808 to (490.56, 509.44, 5.6) mm, rotated rx 0 ry 90 rz 0 deg; joints [-13.07, -27.005, 111.905, -17.055, -84.26, 50.722]
  Set speed (120.0 mm/s)
  MoveL 2809 to (507.59, 498.34, 5.6) mm, rotated rx 0 ry 90 rz 0 deg; joints [-11.712, -26.748, 110.17, -15.736, -82.804, 51.009]
  Set speed (1000.0 mm/s)
  MoveL 2810 to (507.66, 498.41, 5.6) mm, rotated rx 0 ry 90 rz 0 deg; joints [-11.717, -26.746, 110.16, -15.742, -82.796, 51.011]
  Set speed (15.0 mm/s)
  Call Extruder(0.072)
  MoveL 2811 to (507.66, 500.89, 5.6) mm, rotated rx 0 ry 90 rz 0 deg; joints [-11.942, -26.736, 110.097, -15.97, -82.753, 51.051]
  Call Extruder(0.057)
  MoveL 2812 to (509.6, 500.89, 5.6) mm, rotated rx 0 ry 90 rz 0 deg; joints [-11.905, -26.699, 109.864, -15.939, -82.563, 51.101]
  Call Extruder(0.253)
  MoveL 2813 to (509.6, 509.6, 5.6) mm, rotated rx 0 ry 90 rz 0 deg; joints [-12.688, -26.662, 109.636, -16.736, -82.406, 51.247]
  Call Extruder(0.559)
  MoveL 2814 to (490.4, 509.6, 5.6) mm, rotated rx 0 ry 90 rz 0 deg; joints [-13.088, -27.007, 111.919, -17.073, -84.272, 50.72]
  MoveL 2815 to (490.4, 490.4, 5.6) mm, rotated rx 0 ry 90 rz 0 deg; joints [-11.303, -27.074, 112.408, -15.269, -84.635, 50.456]
  Call Extruder(0.154)
  MoveL 2816 to (495.68, 490.4, 5.6) mm, rotated rx 0 ry 90 rz 0 deg; joints [-11.205, -26.988, 111.783, -15.184, -84.113, 50.59]
  Call Extruder(0.055)
  MoveL 2817 to (495.68, 492.29, 5.6) mm, rotated rx 0 ry 90 rz 0 deg; joints [-11.381, -26.982, 111.738, -15.362, -84.08, 50.616]
  Call Extruder(0.062)
  MoveL 2818 to (497.81, 492.29, 5.6) mm, rotated rx 0 ry 90 rz 0 deg; joints [-11.341, -26.946, 111.485, -15.328, -83.87, 50.67]
  Call Extruder(0.010)
  MoveL 2819 to (498.16, 492.29, 5.6) mm, rotated rx 0 ry 90 rz 0 deg; joints [-11.335, -26.94, 111.444, -15.323, -83.835, 50.679]
  Call Extruder(0.007)
  MoveL 2820 to (498.16, 491.94, 5.6) mm, rotated rx 0 ry 90 rz 0 deg; joints [-11.302, -26.941, 111.452, -15.29, -83.841, 50.674]
  Call Extruder(0.045)
  MoveL 2821 to (498.16, 490.4, 5.6) mm, rotated rx 0 ry 90 rz 0 deg; joints [-11.16, -26.947, 111.488, -15.146, -83.868, 50.652]
  Call Extruder(0.083)
  MoveL 2822 to (501, 490.4, 5.6) mm, rotated rx 0 ry 90 rz 0 deg; joints [-11.108, -26.897, 111.151, -15.102, -83.588, 50.723]
  Call Extruder(0.045)
  MoveL 2823 to (500.99, 491.94, 5.6) mm, rotated rx 0 ry 90 rz 0 deg; joints [-11.25, -26.892, 111.114, -15.246, -83.562, 50.745]
  Call Extruder(0.010)
  MoveL 2824 to (500.99, 492.29, 5.6) mm, rotated rx 0 ry 90 rz 0 deg; joints [-11.283, -26.891, 111.106, -15.279, -83.556, 50.75]
  Call Extruder(0.007)
  MoveL 2825 to (501.34, 492.29, 5.6) mm, rotated rx 0 ry 90 rz 0 deg; joints [-11.276, -26.885, 111.064, -15.273, -83.522, 50.759]
  Call Extruder(0.064)
  MoveL 2826 to (503.53, 492.29, 5.6) mm, rotated rx 0 ry 90 rz 0 deg; joints [-11.236, -26.845, 110.803, -15.24, -83.306, 50.814]
  Call Extruder(0.055)
  MoveL 2827 to (503.53, 490.4, 5.6) mm, rotated rx 0 ry 90 rz 0 deg; joints [-11.063, -26.852, 110.847, -15.064, -83.338, 50.786]
  Call Extruder(0.177)
  MoveL 2828 to (509.6, 490.4, 5.6) mm, rotated rx 0 ry 90 rz 0 deg; joints [-10.955, -26.74, 110.119, -14.975, -82.74, 50.935]
  Call Extruder(0.233)
  MoveL 2829 to (509.6, 498.41, 5.6) mm, rotated rx 0 ry 90 rz 0 deg; joints [-11.681, -26.709, 109.926, -15.712, -82.606, 51.061]
  Call Extruder(0.057)
  MoveL 2830 to (507.66, 498.41, 5.6) mm, rotated rx 0 ry 90 rz 0 deg; joints [-11.717, -26.746, 110.16, -15.742, -82.796, 51.011]
  Set speed (120.0 mm/s)
  MoveL 2831 to (507.66, 498.81, 5.6) mm, rotated rx 0 ry 90 rz 0 deg; joints [-11.753, -26.744, 110.15, -15.778, -82.789, 51.018]
  Set speed (1000.0 mm/s)
  MoveL 2832 to (506.96, 498.81, 5.6) mm, rotated rx 0 ry 90 rz 0 deg; joints [-11.766, -26.758, 110.234, -15.789, -82.858, 51]
  Set speed (1000.0 mm/s)
  MoveL 2833 to (490.68, 490.68, 5.6) mm, rotated rx 0 ry 90 rz 0 deg; joints [-11.324, -27.069, 112.368, -15.291, -84.603, 50.466]
  Set speed (1000.0 mm/s)
  MoveL 2834 to (490.68, 490.68, 5.7) mm, rotated rx 0 ry 90 rz 0 deg; joints [-11.324, -27.079, 112.373, -15.291, -84.598, 50.468]
  Set speed (30.0 mm/s)
  Call Extruder(0.767)
  MoveL 2835 to (509.32, 509.32, 5.7) mm, rotated rx 0 ry 90 rz 0 deg; joints [-12.669, -26.679, 109.682, -16.715, -82.434, 51.236]
  MoveL 2836 to (509.44, 509.44, 5.7) mm, rotated rx 0 ry 90 rz 0 deg; joints [-12.677, -26.676, 109.664, -16.725, -82.419, 51.241]
  Set speed (120.0 mm/s)
  MoveL 2837 to (508.73, 501.17, 5.7) mm, rotated rx 0 ry 90 rz 0 deg; joints [-11.946, -26.725, 109.967, -15.979, -82.638, 51.085]
  Set speed (30.0 mm/s)
  Call Extruder(0.335)
  MoveL 2838 to (500.58, 509.32, 5.7) mm, rotated rx 0 ry 90 rz 0 deg; joints [-12.847, -26.844, 110.727, -16.864, -83.282, 50.999]
  Set speed (120.0 mm/s)
  MoveL 2839 to (499.42, 509.32, 5.7) mm, rotated rx 0 ry 90 rz 0 deg; joints [-12.872, -26.865, 110.865, -16.884, -83.395, 50.968]
  Set speed (30.0 mm/s)
  Call Extruder(0.360)
  MoveL 2840 to (490.68, 500.58, 5.7) mm, rotated rx 0 ry 90 rz 0 deg; joints [-12.247, -27.046, 112.13, -16.223, -84.416, 50.6]
  Set speed (120.0 mm/s)
  MoveL 2841 to (490.68, 499.42, 5.7) mm, rotated rx 0 ry 90 rz 0 deg; joints [-12.139, -27.05, 112.159, -16.114, -84.438, 50.584]
  Set speed (30.0 mm/s)
  Call Extruder(0.282)
  MoveL 2842 to (497.53, 492.57, 5.7) mm, rotated rx 0 ry 90 rz 0 deg; joints [-11.372, -26.961, 111.518, -15.359, -83.888, 50.668]
  Set speed (120.0 mm/s)
  MoveL 2843 to (498.5, 491.6, 5.7) mm, rotated rx 0 ry 90 rz 0 deg; joints [-11.264, -26.947, 111.425, -15.253, -83.809, 50.679]
  Set speed (30.0 mm/s)
  Call Extruder(0.038)
  MoveL 2844 to (499.42, 490.68, 5.7) mm, rotated rx 0 ry 90 rz 0 deg; joints [-11.163, -26.935, 111.337, -15.152, -83.734, 50.689]
  Set speed (120.0 mm/s)
  MoveL 2845 to (500.91, 492.32, 5.7) mm, rotated rx 0 ry 90 rz 0 deg; joints [-11.287, -26.903, 111.121, -15.283, -83.559, 50.75]
  Set speed (1000.0 mm/s)
  MoveL 2846 to (502.47, 492.57, 5.7) mm, rotated rx 0 ry 90 rz 0 deg; joints [-11.281, -26.874, 110.928, -15.282, -83.401, 50.793]
  Set speed (30.0 mm/s)
  Call Extruder(0.229)
  MoveL 2847 to (508.03, 498.13, 5.7) mm, rotated rx 0 ry 90 rz 0 deg; joints [-11.685, -26.751, 110.128, -15.71, -82.76, 51.018]
  MoveL 2848 to (508.15, 498.25, 5.7) mm, rotated rx 0 ry 90 rz 0 deg; joints [-11.693, -26.748, 110.11, -15.72, -82.746, 51.023]
  Set speed (120.0 mm/s)
  MoveL 2849 to (509.32, 490.68, 5.7) mm, rotated rx 0 ry 90 rz 0 deg; joints [-10.985, -26.754, 110.152, -15.005, -82.758, 50.934]
  Set speed (30.0 mm/s)
  Call Extruder(0.767)
  MoveL 2850 to (490.68, 509.32, 5.7) mm, rotated rx 0 ry 90 rz 0 deg; joints [-13.056, -27.015, 111.899, -17.042, -84.245, 50.726]
  MoveL 2851 to (490.56, 509.44, 5.7) mm, rotated rx 0 ry 90 rz 0 deg; joints [-13.07, -27.016, 111.91, -17.055, -84.255, 50.724]
  Set speed (120.0 mm/s)
  MoveL 2852 to (507.59, 498.34, 5.7) mm, rotated rx 0 ry 90 rz 0 deg; joints [-11.712, -26.758, 110.175, -15.736, -82.799, 51.01]
  Set speed (1000.0 mm/s)
  MoveL 2853 to (507.66, 498.41, 5.7) mm, rotated rx 0 ry 90 rz 0 deg; joints [-11.717, -26.756, 110.165, -15.742, -82.791, 51.013]
  Set speed (15.0 mm/s)
  Call Extruder(0.072)
  MoveL 2854 to (507.66, 500.89, 5.7) mm, rotated rx 0 ry 90 rz 0 deg; joints [-11.941, -26.747, 110.103, -15.97, -82.748, 51.052]
  Call Extruder(0.057)
  MoveL 2855 to (509.6, 500.89, 5.7) mm, rotated rx 0 ry 90 rz 0 deg; joints [-11.905, -26.709, 109.869, -15.939, -82.558, 51.103]
  Call Extruder(0.254)
  MoveL 2856 to (509.6, 509.6, 5.7) mm, rotated rx 0 ry 90 rz 0 deg; joints [-12.688, -26.672, 109.641, -16.737, -82.401, 51.248]
  Call Extruder(0.559)
  MoveL 2857 to (490.4, 509.6, 5.7) mm, rotated rx 0 ry 90 rz 0 deg; joints [-13.088, -27.018, 111.924, -17.073, -84.267, 50.722]
  MoveL 2858 to (490.4, 490.4, 5.7) mm, rotated rx 0 ry 90 rz 0 deg; joints [-11.303, -27.085, 112.413, -15.269, -84.63, 50.457]
  Call Extruder(0.155)
  MoveL 2859 to (495.73, 490.4, 5.7) mm, rotated rx 0 ry 90 rz 0 deg; joints [-11.204, -26.998, 111.782, -15.184, -84.103, 50.593]
  Call Extruder(0.055)
  MoveL 2860 to (495.74, 492.29, 5.7) mm, rotated rx 0 ry 90 rz 0 deg; joints [-11.38, -26.992, 111.737, -15.361, -84.07, 50.618]
  Call Extruder(0.072)
  MoveL 2861 to (498.22, 492.29, 5.7) mm, rotated rx 0 ry 90 rz 0 deg; joints [-11.334, -26.95, 111.442, -15.322, -83.825, 50.681]
  Call Extruder(0.055)
  MoveL 2862 to (498.22, 490.4, 5.7) mm, rotated rx 0 ry 90 rz 0 deg; joints [-11.159, -26.956, 111.487, -15.145, -83.857, 50.655]
  Call Extruder(0.079)
  MoveL 2863 to (500.93, 490.4, 5.7) mm, rotated rx 0 ry 90 rz 0 deg; joints [-11.109, -26.909, 111.163, -15.103, -83.589, 50.723]
  Call Extruder(0.055)
  MoveL 2864 to (500.93, 492.29, 5.7) mm, rotated rx 0 ry 90 rz 0 deg; joints [-11.284, -26.902, 111.119, -15.28, -83.557, 50.75]
  Call Extruder(0.074)
  MoveL 2865 to (503.47, 492.29, 5.7) mm, rotated rx 0 ry 90 rz 0 deg; joints [-11.237, -26.857, 110.816, -15.241, -83.307, 50.814]
  Call Extruder(0.055)
  MoveL 2866 to (503.47, 490.4, 5.7) mm, rotated rx 0 ry 90 rz 0 deg; joints [-11.064, -26.864, 110.86, -15.065, -83.339, 50.786]
  Call Extruder(0.178)
  MoveL 2867 to (509.6, 490.4, 5.7) mm, rotated rx 0 ry 90 rz 0 deg; joints [-10.955, -26.75, 110.124, -14.975, -82.735, 50.937]
  Call Extruder(0.233)
  MoveL 2868 to (509.6, 498.41, 5.7) mm, rotated rx 0 ry 90 rz 0 deg; joints [-11.68, -26.719, 109.931, -15.712, -82.601, 51.062]
  Call Extruder(0.057)
  MoveL 2869 to (507.66, 498.41, 5.7) mm, rotated rx 0 ry 90 rz 0 deg; joints [-11.717, -26.756, 110.165, -15.742, -82.791, 51.013]
  Set speed (120.0 mm/s)
  MoveL 2870 to (507.66, 498.81, 5.7) mm, rotated rx 0 ry 90 rz 0 deg; joints [-11.753, -26.755, 110.155, -15.778, -82.784, 51.019]
  Set speed (1000.0 mm/s)
  MoveL 2871 to (506.96, 498.81, 5.7) mm, rotated rx 0 ry 90 rz 0 deg; joints [-11.766, -26.768, 110.239, -15.789, -82.853, 51.001]
  Set speed (1000.0 mm/s)
  MoveL 2872 to (490.68, 490.68, 5.7) mm, rotated rx 0 ry 90 rz 0 deg; joints [-11.324, -27.079, 112.373, -15.291, -84.598, 50.468]
  Set speed (1000.0 mm/s)
  MoveL 2873 to (490.68, 490.68, 5.8) mm, rotated rx 0 ry 90 rz 0 deg; joints [-11.324, -27.09, 112.379, -15.291, -84.593, 50.469]
  Set speed (30.0 mm/s)
  Call Extruder(0.767)
  MoveL 2874 to (509.32, 509.32, 5.8) mm, rotated rx 0 ry 90 rz 0 deg; joints [-12.669, -26.689, 109.687, -16.716, -82.429, 51.238]
  MoveL 2875 to (509.44, 509.44, 5.8) mm, rotated rx 0 ry 90 rz 0 deg; joints [-12.677, -26.686, 109.669, -16.725, -82.414, 51.243]
  Set speed (120.0 mm/s)
  MoveL 2876 to (508.73, 501.17, 5.8) mm, rotated rx 0 ry 90 rz 0 deg; joints [-11.946, -26.735, 109.972, -15.979, -82.633, 51.086]
  Set speed (30.0 mm/s)
  Call Extruder(0.336)
  MoveL 2877 to (500.58, 509.32, 5.8) mm, rotated rx 0 ry 90 rz 0 deg; joints [-12.847, -26.854, 110.733, -16.864, -83.277, 51.001]
  Set speed (120.0 mm/s)
  MoveL 2878 to (499.42, 509.32, 5.8) mm, rotated rx 0 ry 90 rz 0 deg; joints [-12.872, -26.875, 110.87, -16.884, -83.39, 50.969]
  Set speed (30.0 mm/s)
  Call Extruder(0.360)
  MoveL 2879 to (490.68, 500.58, 5.8) mm, rotated rx 0 ry 90 rz 0 deg; joints [-12.247, -27.057, 112.135, -16.223, -84.411, 50.602]
  Set speed (120.0 mm/s)
  MoveL 2880 to (490.68, 499.42, 5.8) mm, rotated rx 0 ry 90 rz 0 deg; joints [-12.139, -27.061, 112.165, -16.114, -84.433, 50.586]
  Set speed (30.0 mm/s)
  Call Extruder(0.282)
  MoveL 2881 to (497.53, 492.57, 5.8) mm, rotated rx 0 ry 90 rz 0 deg; joints [-11.372, -26.971, 111.523, -15.359, -83.883, 50.669]
  MoveL 2882 to (497.65, 492.45, 5.8) mm, rotated rx 0 ry 90 rz 0 deg; joints [-11.359, -26.97, 111.511, -15.346, -83.873, 50.671]
  Set speed (120.0 mm/s)
  MoveL 2883 to (498.56, 491.54, 5.8) mm, rotated rx 0 ry 90 rz 0 deg; joints [-11.258, -26.957, 111.425, -15.246, -83.799, 50.681]
  Set speed (30.0 mm/s)
  Call Extruder(0.035)
  MoveL 2884 to (499.42, 490.68, 5.8) mm, rotated rx 0 ry 90 rz 0 deg; joints [-11.163, -26.945, 111.343, -15.153, -83.729, 50.69]
  Set speed (120.0 mm/s)
  MoveL 2885 to (500.84, 492.32, 5.8) mm, rotated rx 0 ry 90 rz 0 deg; joints [-11.288, -26.914, 111.134, -15.284, -83.56, 50.75]
  Set speed (1000.0 mm/s)
  MoveL 2886 to (502.47, 492.57, 5.8) mm, rotated rx 0 ry 90 rz 0 deg; joints [-11.281, -26.885, 110.933, -15.282, -83.396, 50.794]
  Set speed (30.0 mm/s)
  Call Extruder(0.229)
  MoveL 2887 to (508.03, 498.13, 5.8) mm, rotated rx 0 ry 90 rz 0 deg; joints [-11.685, -26.761, 110.133, -15.71, -82.755, 51.019]
  MoveL 2888 to (508.15, 498.25, 5.8) mm, rotated rx 0 ry 90 rz 0 deg; joints [-11.693, -26.758, 110.115, -15.72, -82.741, 51.024]
  Set speed (120.0 mm/s)
  MoveL 2889 to (509.32, 490.68, 5.8) mm, rotated rx 0 ry 90 rz 0 deg; joints [-10.985, -26.765, 110.157, -15.005, -82.753, 50.935]
  Set speed (30.0 mm/s)
  Call Extruder(0.767)
  MoveL 2890 to (490.68, 509.32, 5.8) mm, rotated rx 0 ry 90 rz 0 deg; joints [-13.056, -27.025, 111.904, -17.042, -84.24, 50.727]
  MoveL 2891 to (490.56, 509.44, 5.8) mm, rotated rx 0 ry 90 rz 0 deg; joints [-13.07, -27.027, 111.915, -17.055, -84.25, 50.726]
  Set speed (120.0 mm/s)
  MoveL 2892 to (507.59, 498.34, 5.8) mm, rotated rx 0 ry 90 rz 0 deg; joints [-11.712, -26.769, 110.18, -15.736, -82.794, 51.011]
  Set speed (1000.0 mm/s)
  MoveL 2893 to (507.66, 498.41, 5.8) mm, rotated rx 0 ry 90 rz 0 deg; joints [-11.717, -26.767, 110.17, -15.742, -82.786, 51.014]
  Set speed (15.0 mm/s)
  Call Extruder(0.072)
  MoveL 2894 to (507.66, 500.89, 5.8) mm, rotated rx 0 ry 90 rz 0 deg; joints [-11.941, -26.757, 110.108, -15.97, -82.743, 51.054]
  Call Extruder(0.057)
  MoveL 2895 to (509.6, 500.89, 5.8) mm, rotated rx 0 ry 90 rz 0 deg; joints [-11.904, -26.72, 109.874, -15.94, -82.553, 51.104]
  Call Extruder(0.254)
  MoveL 2896 to (509.6, 509.6, 5.8) mm, rotated rx 0 ry 90 rz 0 deg; joints [-12.688, -26.683, 109.646, -16.737, -82.396, 51.25]
  Call Extruder(0.559)
  MoveL 2897 to (490.4, 509.6, 5.8) mm, rotated rx 0 ry 90 rz 0 deg; joints [-13.088, -27.029, 111.929, -17.073, -84.262, 50.723]
  MoveL 2898 to (490.4, 490.4, 5.8) mm, rotated rx 0 ry 90 rz 0 deg; joints [-11.303, -27.095, 112.418, -15.269, -84.625, 50.459]
  Call Extruder(0.157)
  MoveL 2899 to (495.79, 490.4, 5.8) mm, rotated rx 0 ry 90 rz 0 deg; joints [-11.203, -27.008, 111.781, -15.183, -84.092, 50.595]
  Call Extruder(0.055)
  MoveL 2900 to (495.79, 492.29, 5.8) mm, rotated rx 0 ry 90 rz 0 deg; joints [-11.379, -27.001, 111.736, -15.36, -84.059, 50.621]
  Call Extruder(0.062)
  MoveL 2901 to (497.93, 492.29, 5.8) mm, rotated rx 0 ry 90 rz 0 deg; joints [-11.339, -26.965, 111.482, -15.327, -83.848, 50.676]
  Call Extruder(0.010)
  MoveL 2902 to (498.28, 492.29, 5.8) mm, rotated rx 0 ry 90 rz 0 deg; joints [-11.332, -26.959, 111.44, -15.321, -83.814, 50.684]
  Call Extruder(0.007)
  MoveL 2903 to (498.28, 491.94, 5.8) mm, rotated rx 0 ry 90 rz 0 deg; joints [-11.3, -26.96, 111.448, -15.288, -83.82, 50.679]
  Call Extruder(0.045)
  MoveL 2904 to (498.28, 490.4, 5.8) mm, rotated rx 0 ry 90 rz 0 deg; joints [-11.158, -26.966, 111.485, -15.144, -83.846, 50.658]
  Call Extruder(0.076)
  MoveL 2905 to (500.87, 490.4, 5.8) mm, rotated rx 0 ry 90 rz 0 deg; joints [-11.11, -26.921, 111.176, -15.104, -83.59, 50.723]
  Call Extruder(0.045)
  MoveL 2906 to (500.87, 491.94, 5.8) mm, rotated rx 0 ry 90 rz 0 deg; joints [-11.253, -26.915, 111.139, -15.248, -83.564, 50.745]
  Call Extruder(0.010)
  MoveL 2907 to (500.87, 492.29, 5.8) mm, rotated rx 0 ry 90 rz 0 deg; joints [-11.285, -26.914, 111.131, -15.281, -83.558, 50.75]
  Call Extruder(0.007)
  MoveL 2908 to (501.22, 492.29, 5.8) mm, rotated rx 0 ry 90 rz 0 deg; joints [-11.278, -26.908, 111.089, -15.275, -83.523, 50.759]
  Call Extruder(0.064)
  MoveL 2909 to (503.4, 492.29, 5.8) mm, rotated rx 0 ry 90 rz 0 deg; joints [-11.238, -26.869, 110.829, -15.242, -83.309, 50.813]
  Call Extruder(0.055)
  MoveL 2910 to (503.41, 490.4, 5.8) mm, rotated rx 0 ry 90 rz 0 deg; joints [-11.065, -26.875, 110.873, -15.066, -83.34, 50.786]
  Call Extruder(0.180)
  MoveL 2911 to (509.6, 490.4, 5.8) mm, rotated rx 0 ry 90 rz 0 deg; joints [-10.955, -26.761, 110.13, -14.975, -82.73, 50.938]
  Call Extruder(0.233)
  MoveL 2912 to (509.6, 498.41, 5.8) mm, rotated rx 0 ry 90 rz 0 deg; joints [-11.68, -26.73, 109.937, -15.712, -82.596, 51.064]
  Call Extruder(0.057)
  MoveL 2913 to (507.66, 498.41, 5.8) mm, rotated rx 0 ry 90 rz 0 deg; joints [-11.717, -26.767, 110.17, -15.742, -82.786, 51.014]
  Set speed (120.0 mm/s)
  MoveL 2914 to (507.66, 498.81, 5.8) mm, rotated rx 0 ry 90 rz 0 deg; joints [-11.753, -26.765, 110.16, -15.779, -82.779, 51.021]
  Set speed (1000.0 mm/s)
  MoveL 2915 to (506.96, 498.81, 5.8) mm, rotated rx 0 ry 90 rz 0 deg; joints [-11.766, -26.779, 110.244, -15.789, -82.848, 51.003]
  Set speed (1000.0 mm/s)
  MoveL 2916 to (490.68, 490.68, 5.8) mm, rotated rx 0 ry 90 rz 0 deg; joints [-11.324, -27.09, 112.379, -15.291, -84.593, 50.469]
  Set speed (1000.0 mm/s)
  MoveL 2917 to (490.68, 490.68, 5.9) mm, rotated rx 0 ry 90 rz 0 deg; joints [-11.324, -27.101, 112.384, -15.291, -84.587, 50.471]
  Set speed (30.0 mm/s)
  Call Extruder(0.767)
  MoveL 2918 to (509.32, 509.32, 5.9) mm, rotated rx 0 ry 90 rz 0 deg; joints [-12.669, -26.7, 109.693, -16.716, -82.424, 51.239]
  MoveL 2919 to (509.44, 509.44, 5.9) mm, rotated rx 0 ry 90 rz 0 deg; joints [-12.677, -26.697, 109.675, -16.725, -82.41, 51.244]
  Set speed (120.0 mm/s)
  MoveL 2920 to (508.73, 501.17, 5.9) mm, rotated rx 0 ry 90 rz 0 deg; joints [-11.946, -26.746, 109.977, -15.979, -82.628, 51.088]
  Set speed (30.0 mm/s)
  Call Extruder(0.336)
  MoveL 2921 to (500.58, 509.32, 5.9) mm, rotated rx 0 ry 90 rz 0 deg; joints [-12.847, -26.865, 110.738, -16.864, -83.272, 51.003]
  Set speed (120.0 mm/s)
  MoveL 2922 to (499.42, 509.32, 5.9) mm, rotated rx 0 ry 90 rz 0 deg; joints [-12.872, -26.886, 110.876, -16.884, -83.385, 50.971]
  Set speed (30.0 mm/s)
  Call Extruder(0.360)
  MoveL 2923 to (490.68, 500.58, 5.9) mm, rotated rx 0 ry 90 rz 0 deg; joints [-12.247, -27.068, 112.141, -16.223, -84.406, 50.603]
  Set speed (120.0 mm/s)
  MoveL 2924 to (490.68, 499.42, 5.9) mm, rotated rx 0 ry 90 rz 0 deg; joints [-12.139, -27.072, 112.17, -16.114, -84.428, 50.587]
  Set speed (30.0 mm/s)
  Call Extruder(0.282)
  MoveL 2925 to (497.53, 492.57, 5.9) mm, rotated rx 0 ry 90 rz 0 deg; joints [-11.372, -26.982, 111.528, -15.359, -83.878, 50.671]
  MoveL 2926 to (497.65, 492.45, 5.9) mm, rotated rx 0 ry 90 rz 0 deg; joints [-11.359, -26.98, 111.517, -15.346, -83.868, 50.672]
  Set speed (120.0 mm/s)
  MoveL 2927 to (498.62, 491.48, 5.9) mm, rotated rx 0 ry 90 rz 0 deg; joints [-11.251, -26.967, 111.424, -15.24, -83.789, 50.683]
  Set speed (30.0 mm/s)
  Call Extruder(0.033)
  MoveL 2928 to (499.42, 490.68, 5.9) mm, rotated rx 0 ry 90 rz 0 deg; joints [-11.163, -26.956, 111.348, -15.153, -83.724, 50.692]
  Set speed (120.0 mm/s)
  MoveL 2929 to (500.78, 492.32, 5.9) mm, rotated rx 0 ry 90 rz 0 deg; joints [-11.289, -26.926, 111.146, -15.285, -83.561, 50.749]
  Set speed (1000.0 mm/s)
  MoveL 2930 to (502.47, 492.57, 5.9) mm, rotated rx 0 ry 90 rz 0 deg; joints [-11.281, -26.895, 110.939, -15.282, -83.391, 50.795]
  Set speed (30.0 mm/s)
  Call Extruder(0.229)
  MoveL 2931 to (508.02, 498.13, 5.9) mm, rotated rx 0 ry 90 rz 0 deg; joints [-11.684, -26.772, 110.138, -15.71, -82.75, 51.021]
  MoveL 2932 to (508.15, 498.25, 5.9) mm, rotated rx 0 ry 90 rz 0 deg; joints [-11.693, -26.769, 110.121, -15.72, -82.736, 51.026]
  Set speed (120.0 mm/s)
  MoveL 2933 to (509.32, 490.68, 5.9) mm, rotated rx 0 ry 90 rz 0 deg; joints [-10.985, -26.775, 110.162, -15.005, -82.748, 50.937]
  Set speed (30.0 mm/s)
  Call Extruder(0.767)
  MoveL 2934 to (490.68, 509.32, 5.9) mm, rotated rx 0 ry 90 rz 0 deg; joints [-13.056, -27.036, 111.909, -17.042, -84.235, 50.729]
  MoveL 2935 to (490.56, 509.44, 5.9) mm, rotated rx 0 ry 90 rz 0 deg; joints [-13.07, -27.037, 111.921, -17.056, -84.245, 50.727]
  Set speed (120.0 mm/s)
  MoveL 2936 to (507.59, 498.34, 5.9) mm, rotated rx 0 ry 90 rz 0 deg; joints [-11.712, -26.779, 110.186, -15.736, -82.789, 51.013]
  Set speed (1000.0 mm/s)
  MoveL 2937 to (507.66, 498.41, 5.9) mm, rotated rx 0 ry 90 rz 0 deg; joints [-11.717, -26.777, 110.176, -15.742, -82.781, 51.016]
  Set speed (15.0 mm/s)
  Call Extruder(0.072)
  MoveL 2938 to (507.66, 500.89, 5.9) mm, rotated rx 0 ry 90 rz 0 deg; joints [-11.941, -26.768, 110.113, -15.97, -82.738, 51.055]
  Call Extruder(0.057)
  MoveL 2939 to (509.6, 500.89, 5.9) mm, rotated rx 0 ry 90 rz 0 deg; joints [-11.904, -26.73, 109.88, -15.94, -82.548, 51.105]
  Call Extruder(0.254)
  MoveL 2940 to (509.6, 509.6, 5.9) mm, rotated rx 0 ry 90 rz 0 deg; joints [-12.688, -26.693, 109.651, -16.737, -82.391, 51.251]
  Call Extruder(0.559)
  MoveL 2941 to (490.4, 509.6, 5.9) mm, rotated rx 0 ry 90 rz 0 deg; joints [-13.088, -27.039, 111.935, -17.073, -84.257, 50.725]
  MoveL 2942 to (490.4, 490.4, 5.9) mm, rotated rx 0 ry 90 rz 0 deg; joints [-11.303, -27.106, 112.424, -15.269, -84.62, 50.46]
  Call Extruder(0.158)
  MoveL 2943 to (495.84, 490.4, 5.9) mm, rotated rx 0 ry 90 rz 0 deg; joints [-11.202, -27.018, 111.78, -15.182, -84.082, 50.598]
  Call Extruder(0.055)
  MoveL 2944 to (495.85, 492.29, 5.9) mm, rotated rx 0 ry 90 rz 0 deg; joints [-11.378, -27.011, 111.734, -15.36, -84.048, 50.624]
  Call Extruder(0.062)
  MoveL 2945 to (497.99, 492.29, 5.9) mm, rotated rx 0 ry 90 rz 0 deg; joints [-11.338, -26.975, 111.48, -15.326, -83.837, 50.678]
  Call Extruder(0.010)
  MoveL 2946 to (498.34, 492.29, 5.9) mm, rotated rx 0 ry 90 rz 0 deg; joints [-11.331, -26.969, 111.438, -15.32, -83.803, 50.687]
  Call Extruder(0.007)
  MoveL 2947 to (498.34, 491.94, 5.9) mm, rotated rx 0 ry 90 rz 0 deg; joints [-11.299, -26.97, 111.447, -15.288, -83.809, 50.682]
  Call Extruder(0.045)
  MoveL 2948 to (498.34, 490.4, 5.9) mm, rotated rx 0 ry 90 rz 0 deg; joints [-11.156, -26.975, 111.483, -15.143, -83.835, 50.661]
  Call Extruder(0.072)
  MoveL 2949 to (500.81, 490.4, 5.9) mm, rotated rx 0 ry 90 rz 0 deg; joints [-11.112, -26.932, 111.188, -15.105, -83.591, 50.723]
  Call Extruder(0.045)
  MoveL 2950 to (500.81, 491.94, 5.9) mm, rotated rx 0 ry 90 rz 0 deg; joints [-11.254, -26.927, 111.152, -15.249, -83.565, 50.745]
  Call Extruder(0.010)
  MoveL 2951 to (500.81, 492.29, 5.9) mm, rotated rx 0 ry 90 rz 0 deg; joints [-11.286, -26.926, 111.144, -15.282, -83.559, 50.75]
  Call Extruder(0.007)
  MoveL 2952 to (501.16, 492.29, 5.9) mm, rotated rx 0 ry 90 rz 0 deg; joints [-11.279, -26.919, 111.102, -15.276, -83.524, 50.759]
  Call Extruder(0.063)
  MoveL 2953 to (503.34, 492.29, 5.9) mm, rotated rx 0 ry 90 rz 0 deg; joints [-11.24, -26.88, 110.841, -15.243, -83.31, 50.813]
  Call Extruder(0.055)
  MoveL 2954 to (503.34, 490.4, 5.9) mm, rotated rx 0 ry 90 rz 0 deg; joints [-11.066, -26.887, 110.886, -15.067, -83.341, 50.786]
  Call Extruder(0.182)
  MoveL 2955 to (509.6, 490.4, 5.9) mm, rotated rx 0 ry 90 rz 0 deg; joints [-10.955, -26.771, 110.135, -14.975, -82.725, 50.939]
  Call Extruder(0.233)
  MoveL 2956 to (509.6, 498.41, 5.9) mm, rotated rx 0 ry 90 rz 0 deg; joints [-11.68, -26.74, 109.942, -15.712, -82.591, 51.065]
  Call Extruder(0.057)
  MoveL 2957 to (507.66, 498.41, 5.9) mm, rotated rx 0 ry 90 rz 0 deg; joints [-11.717, -26.777, 110.176, -15.742, -82.781, 51.016]
  Set speed (120.0 mm/s)
  MoveL 2958 to (507.66, 498.81, 5.9) mm, rotated rx 0 ry 90 rz 0 deg; joints [-11.753, -26.776, 110.166, -15.779, -82.774, 51.022]
  Set speed (1000.0 mm/s)
  MoveL 2959 to (506.96, 498.81, 5.9) mm, rotated rx 0 ry 90 rz 0 deg; joints [-11.766, -26.789, 110.25, -15.79, -82.843, 51.004]
  Set speed (1000.0 mm/s)
  MoveL 2960 to (490.68, 490.68, 5.9) mm, rotated rx 0 ry 90 rz 0 deg; joints [-11.324, -27.101, 112.384, -15.291, -84.587, 50.471]
  Set speed (1000.0 mm/s)
  MoveL 2961 to (490.68, 490.68, 6) mm, rotated rx 0 ry 90 rz 0 deg; joints [-11.324, -27.111, 112.389, -15.291, -84.582, 50.472]
  Set speed (30.0 mm/s)
  Call Extruder(0.767)
  MoveL 2962 to (509.32, 509.32, 6) mm, rotated rx 0 ry 90 rz 0 deg; joints [-12.669, -26.71, 109.698, -16.716, -82.419, 51.241]
  MoveL 2963 to (509.44, 509.44, 6) mm, rotated rx 0 ry 90 rz 0 deg; joints [-12.677, -26.707, 109.68, -16.725, -82.405, 51.246]
  Set speed (120.0 mm/s)
  MoveL 2964 to (508.73, 501.17, 6) mm, rotated rx 0 ry 90 rz 0 deg; joints [-11.946, -26.756, 109.982, -15.979, -82.623, 51.089]
  Set speed (30.0 mm/s)
  Call Extruder(0.336)
  MoveL 2965 to (500.58, 509.32, 6) mm, rotated rx 0 ry 90 rz 0 deg; joints [-12.847, -26.875, 110.743, -16.864, -83.267, 51.004]
  Set speed (120.0 mm/s)
  MoveL 2966 to (499.42, 509.32, 6) mm, rotated rx 0 ry 90 rz 0 deg; joints [-12.872, -26.896, 110.881, -16.884, -83.38, 50.972]
  Set speed (30.0 mm/s)
  Call Extruder(0.360)
  MoveL 2967 to (490.68, 500.58, 6) mm, rotated rx 0 ry 90 rz 0 deg; joints [-12.247, -27.078, 112.146, -16.223, -84.401, 50.605]
  Set speed (120.0 mm/s)
  MoveL 2968 to (490.68, 499.42, 6) mm, rotated rx 0 ry 90 rz 0 deg; joints [-12.139, -27.082, 112.175, -16.114, -84.423, 50.589]
  Set speed (30.0 mm/s)
  Call Extruder(0.282)
  MoveL 2969 to (497.52, 492.57, 6) mm, rotated rx 0 ry 90 rz 0 deg; joints [-11.372, -26.992, 111.534, -15.359, -83.873, 50.672]
  MoveL 2970 to (497.65, 492.45, 6) mm, rotated rx 0 ry 90 rz 0 deg; joints [-11.359, -26.991, 111.522, -15.346, -83.863, 50.673]
  Set speed (120.0 mm/s)
  MoveL 2971 to (498.68, 491.42, 6) mm, rotated rx 0 ry 90 rz 0 deg; joints [-11.245, -26.977, 111.424, -15.234, -83.779, 50.685]
  Set speed (30.0 mm/s)
  Call Extruder(0.031)
  MoveL 2972 to (499.42, 490.68, 6) mm, rotated rx 0 ry 90 rz 0 deg; joints [-11.163, -26.966, 111.353, -15.153, -83.719, 50.693]
  Set speed (120.0 mm/s)
  MoveL 2973 to (500.72, 492.32, 6) mm, rotated rx 0 ry 90 rz 0 deg; joints [-11.29, -26.938, 111.159, -15.286, -83.562, 50.749]
  Set speed (1000.0 mm/s)
  MoveL 2974 to (502.47, 492.57, 6) mm, rotated rx 0 ry 90 rz 0 deg; joints [-11.281, -26.906, 110.944, -15.283, -83.385, 50.797]
  Set speed (30.0 mm/s)
  Call Extruder(0.228)
  MoveL 2975 to (508.02, 498.12, 6) mm, rotated rx 0 ry 90 rz 0 deg; joints [-11.684, -26.782, 110.144, -15.71, -82.745, 51.022]
  MoveL 2976 to (508.15, 498.25, 6) mm, rotated rx 0 ry 90 rz 0 deg; joints [-11.693, -26.779, 110.126, -15.72, -82.731, 51.027]
  Set speed (120.0 mm/s)
  MoveL 2977 to (509.32, 490.68, 6) mm, rotated rx 0 ry 90 rz 0 deg; joints [-10.985, -26.786, 110.168, -15.005, -82.743, 50.938]
  Set speed (30.0 mm/s)
  Call Extruder(0.767)
  MoveL 2978 to (490.68, 509.32, 6) mm, rotated rx 0 ry 90 rz 0 deg; joints [-13.056, -27.046, 111.915, -17.042, -84.23, 50.73]
  MoveL 2979 to (490.56, 509.44, 6) mm, rotated rx 0 ry 90 rz 0 deg; joints [-13.07, -27.048, 111.926, -17.056, -84.24, 50.729]
  Set speed (120.0 mm/s)
  MoveL 2980 to (507.59, 498.33, 6) mm, rotated rx 0 ry 90 rz 0 deg; joints [-11.712, -26.79, 110.191, -15.737, -82.784, 51.014]
  Set speed (1000.0 mm/s)
  MoveL 2981 to (507.66, 498.41, 6) mm, rotated rx 0 ry 90 rz 0 deg; joints [-11.717, -26.788, 110.181, -15.742, -82.776, 51.017]
  Set speed (15.0 mm/s)
  Call Extruder(0.072)
  MoveL 2982 to (507.66, 500.88, 6) mm, rotated rx 0 ry 90 rz 0 deg; joints [-11.941, -26.778, 110.118, -15.97, -82.733, 51.057]
  Call Extruder(0.057)
  MoveL 2983 to (509.6, 500.89, 6) mm, rotated rx 0 ry 90 rz 0 deg; joints [-11.904, -26.741, 109.885, -15.94, -82.543, 51.107]
  Call Extruder(0.254)
  MoveL 2984 to (509.6, 509.6, 6) mm, rotated rx 0 ry 90 rz 0 deg; joints [-12.688, -26.703, 109.657, -16.737, -82.386, 51.253]
  Call Extruder(0.559)
  MoveL 2985 to (490.4, 509.6, 6) mm, rotated rx 0 ry 90 rz 0 deg; joints [-13.088, -27.05, 111.94, -17.073, -84.252, 50.727]
  MoveL 2986 to (490.4, 490.4, 6) mm, rotated rx 0 ry 90 rz 0 deg; joints [-11.303, -27.117, 112.429, -15.269, -84.615, 50.461]
  Call Extruder(0.160)
  MoveL 2987 to (495.9, 490.4, 6) mm, rotated rx 0 ry 90 rz 0 deg; joints [-11.201, -27.027, 111.778, -15.181, -84.071, 50.601]
  Call Extruder(0.055)
  MoveL 2988 to (495.9, 492.29, 6) mm, rotated rx 0 ry 90 rz 0 deg; joints [-11.377, -27.021, 111.733, -15.359, -84.038, 50.627]
  Call Extruder(0.062)
  MoveL 2989 to (498.05, 492.29, 6) mm, rotated rx 0 ry 90 rz 0 deg; joints [-11.337, -26.984, 111.478, -15.325, -83.826, 50.681]
  Call Extruder(0.010)
  MoveL 2990 to (498.4, 492.29, 6) mm, rotated rx 0 ry 90 rz 0 deg; joints [-11.33, -26.978, 111.437, -15.319, -83.792, 50.69]
  Call Extruder(0.007)
  MoveL 2991 to (498.4, 491.94, 6) mm, rotated rx 0 ry 90 rz 0 deg; joints [-11.298, -26.98, 111.445, -15.287, -83.798, 50.685]
  Call Extruder(0.035)
  MoveL 2992 to (498.4, 490.75, 6) mm, rotated rx 0 ry 90 rz 0 deg; joints [-11.188, -26.984, 111.473, -15.175, -83.818, 50.669]
  Call Extruder(0.010)
  MoveL 2993 to (498.4, 490.4, 6) mm, rotated rx 0 ry 90 rz 0 deg; joints [-11.155, -26.985, 111.481, -15.143, -83.824, 50.664]
  Call Extruder(0.007)
  MoveL 2994 to (498.75, 490.4, 6) mm, rotated rx 0 ry 90 rz 0 deg; joints [-11.149, -26.979, 111.44, -15.137, -83.79, 50.672]
  Call Extruder(0.058)
  MoveL 2995 to (500.75, 490.4, 6) mm, rotated rx 0 ry 90 rz 0 deg; joints [-11.113, -26.944, 111.201, -15.107, -83.592, 50.723]
  Call Extruder(0.045)
  MoveL 2996 to (500.75, 491.94, 6) mm, rotated rx 0 ry 90 rz 0 deg; joints [-11.255, -26.939, 111.165, -15.25, -83.566, 50.745]
  Call Extruder(0.010)
  MoveL 2997 to (500.75, 492.29, 6) mm, rotated rx 0 ry 90 rz 0 deg; joints [-11.287, -26.937, 111.156, -15.283, -83.56, 50.75]
  Call Extruder(0.007)
  MoveL 2998 to (501.1, 492.29, 6) mm, rotated rx 0 ry 90 rz 0 deg; joints [-11.281, -26.931, 111.115, -15.278, -83.525, 50.758]
  Call Extruder(0.063)
  MoveL 2999 to (503.28, 492.29, 6) mm, rotated rx 0 ry 90 rz 0 deg; joints [-11.241, -26.892, 110.854, -15.244, -83.311, 50.813]
  Call Extruder(0.055)
  MoveL 3000 to (503.28, 490.4, 6) mm, rotated rx 0 ry 90 rz 0 deg; joints [-11.067, -26.899, 110.899, -15.068, -83.342, 50.785]
  Call Extruder(0.184)
  MoveL 3001 to (509.6, 490.4, 6) mm, rotated rx 0 ry 90 rz 0 deg; joints [-10.955, -26.781, 110.14, -14.976, -82.72, 50.941]
  Call Extruder(0.233)
  MoveL 3002 to (509.6, 498.4, 6) mm, rotated rx 0 ry 90 rz 0 deg; joints [-11.68, -26.751, 109.947, -15.712, -82.586, 51.067]
  Call Extruder(0.057)
  MoveL 3003 to (507.66, 498.41, 6) mm, rotated rx 0 ry 90 rz 0 deg; joints [-11.717, -26.788, 110.181, -15.742, -82.776, 51.017]
  Set speed (120.0 mm/s)
  MoveL 3004 to (507.66, 498.81, 6) mm, rotated rx 0 ry 90 rz 0 deg; joints [-11.753, -26.786, 110.171, -15.779, -82.769, 51.023]
  Set speed (1000.0 mm/s)
  MoveL 3005 to (506.96, 498.81, 6) mm, rotated rx 0 ry 90 rz 0 deg; joints [-11.766, -26.8, 110.255, -15.79, -82.838, 51.005]
  Set speed (1000.0 mm/s)
  MoveL 3006 to (490.68, 490.68, 6) mm, rotated rx 0 ry 90 rz 0 deg; joints [-11.324, -27.111, 112.389, -15.291, -84.582, 50.472]
  Set speed (1000.0 mm/s)
  MoveL 3007 to (490.68, 490.68, 6.1) mm, rotated rx 0 ry 90 rz 0 deg; joints [-11.324, -27.122, 112.395, -15.291, -84.577, 50.474]
  Set speed (30.0 mm/s)
  Call Extruder(0.767)
  MoveL 3008 to (509.32, 509.32, 6.1) mm, rotated rx 0 ry 90 rz 0 deg; joints [-12.669, -26.721, 109.703, -16.716, -82.414, 51.242]
  MoveL 3009 to (509.44, 509.44, 6.1) mm, rotated rx 0 ry 90 rz 0 deg; joints [-12.677, -26.718, 109.685, -16.725, -82.4, 51.247]
  Set speed (120.0 mm/s)
  MoveL 3010 to (508.73, 501.16, 6.1) mm, rotated rx 0 ry 90 rz 0 deg; joints [-11.946, -26.767, 109.987, -15.979, -82.618, 51.09]
  Set speed (30.0 mm/s)
  Call Extruder(0.336)
  MoveL 3011 to (500.58, 509.32, 6.1) mm, rotated rx 0 ry 90 rz 0 deg; joints [-12.847, -26.886, 110.748, -16.864, -83.262, 51.006]
  Set speed (120.0 mm/s)
  MoveL 3012 to (499.42, 509.32, 6.1) mm, rotated rx 0 ry 90 rz 0 deg; joints [-12.872, -26.907, 110.886, -16.885, -83.375, 50.974]
  Set speed (30.0 mm/s)
  Call Extruder(0.360)
  MoveL 3013 to (490.68, 500.58, 6.1) mm, rotated rx 0 ry 90 rz 0 deg; joints [-12.247, -27.089, 112.151, -16.223, -84.396, 50.606]
  Set speed (120.0 mm/s)
  MoveL 3014 to (490.68, 499.42, 6.1) mm, rotated rx 0 ry 90 rz 0 deg; joints [-12.139, -27.093, 112.181, -16.115, -84.418, 50.59]
  Set speed (30.0 mm/s)
  Call Extruder(0.282)
  MoveL 3015 to (497.52, 492.57, 6.1) mm, rotated rx 0 ry 90 rz 0 deg; joints [-11.372, -27.003, 111.539, -15.36, -83.868, 50.673]
  MoveL 3016 to (497.65, 492.45, 6.1) mm, rotated rx 0 ry 90 rz 0 deg; joints [-11.359, -27.001, 111.527, -15.346, -83.858, 50.675]
  Set speed (120.0 mm/s)
  MoveL 3017 to (498.74, 491.36, 6.1) mm, rotated rx 0 ry 90 rz 0 deg; joints [-11.238, -26.986, 111.424, -15.228, -83.769, 50.687]
  Set speed (30.0 mm/s)
  Call Extruder(0.028)
  MoveL 3018 to (499.42, 490.68, 6.1) mm, rotated rx 0 ry 90 rz 0 deg; joints [-11.163, -26.977, 111.359, -15.153, -83.714, 50.695]
  Set speed (120.0 mm/s)
  MoveL 3019 to (500.66, 492.32, 6.1) mm, rotated rx 0 ry 90 rz 0 deg; joints [-11.291, -26.949, 111.172, -15.287, -83.563, 50.749]
  Set speed (1000.0 mm/s)
  MoveL 3020 to (502.47, 492.57, 6.1) mm, rotated rx 0 ry 90 rz 0 deg; joints [-11.281, -26.916, 110.949, -15.283, -83.38, 50.798]
  Set speed (30.0 mm/s)
  Call Extruder(0.228)
  MoveL 3021 to (508.02, 498.12, 6.1) mm, rotated rx 0 ry 90 rz 0 deg; joints [-11.684, -26.793, 110.149, -15.71, -82.74, 51.023]
  MoveL 3022 to (508.14, 498.25, 6.1) mm, rotated rx 0 ry 90 rz 0 deg; joints [-11.693, -26.79, 110.132, -15.72, -82.726, 51.028]
  Set speed (120.0 mm/s)
  MoveL 3023 to (509.32, 490.68, 6.1) mm, rotated rx 0 ry 90 rz 0 deg; joints [-10.985, -26.796, 110.173, -15.006, -82.738, 50.94]
  Set speed (30.0 mm/s)
  Call Extruder(0.767)
  MoveL 3024 to (490.68, 509.32, 6.1) mm, rotated rx 0 ry 90 rz 0 deg; joints [-13.056, -27.057, 111.92, -17.042, -84.225, 50.732]
  MoveL 3025 to (490.56, 509.44, 6.1) mm, rotated rx 0 ry 90 rz 0 deg; joints [-13.07, -27.059, 111.931, -17.056, -84.235, 50.73]
  Set speed (120.0 mm/s)
  MoveL 3026 to (507.59, 498.33, 6.1) mm, rotated rx 0 ry 90 rz 0 deg; joints [-11.711, -26.8, 110.196, -15.737, -82.779, 51.016]
  Set speed (1000.0 mm/s)
  MoveL 3027 to (507.66, 498.4, 6.1) mm, rotated rx 0 ry 90 rz 0 deg; joints [-11.716, -26.798, 110.186, -15.742, -82.771, 51.018]
  Set speed (15.0 mm/s)
  Call Extruder(0.072)
  MoveL 3028 to (507.66, 500.88, 6.1) mm, rotated rx 0 ry 90 rz 0 deg; joints [-11.941, -26.788, 110.124, -15.97, -82.728, 51.058]
  Call Extruder(0.057)
  MoveL 3029 to (509.6, 500.89, 6.1) mm, rotated rx 0 ry 90 rz 0 deg; joints [-11.904, -26.751, 109.89, -15.94, -82.538, 51.108]
  Call Extruder(0.254)
  MoveL 3030 to (509.6, 509.6, 6.1) mm, rotated rx 0 ry 90 rz 0 deg; joints [-12.688, -26.714, 109.662, -16.737, -82.381, 51.254]
  Call Extruder(0.559)
  MoveL 3031 to (490.4, 509.6, 6.1) mm, rotated rx 0 ry 90 rz 0 deg; joints [-13.088, -27.061, 111.945, -17.074, -84.247, 50.728]
  MoveL 3032 to (490.4, 490.4, 6.1) mm, rotated rx 0 ry 90 rz 0 deg; joints [-11.303, -27.127, 112.434, -15.269, -84.61, 50.463]
  Call Extruder(0.162)
  MoveL 3033 to (495.95, 490.4, 6.1) mm, rotated rx 0 ry 90 rz 0 deg; joints [-11.2, -27.037, 111.777, -15.181, -84.06, 50.604]
  Call Extruder(0.055)
  MoveL 3034 to (495.96, 492.29, 6.1) mm, rotated rx 0 ry 90 rz 0 deg; joints [-11.376, -27.031, 111.732, -15.358, -84.027, 50.63]
  Call Extruder(0.063)
  MoveL 3035 to (498.11, 492.29, 6.1) mm, rotated rx 0 ry 90 rz 0 deg; joints [-11.336, -26.994, 111.476, -15.324, -83.815, 50.684]
  Call Extruder(0.010)
  MoveL 3036 to (498.46, 492.29, 6.1) mm, rotated rx 0 ry 90 rz 0 deg; joints [-11.329, -26.988, 111.435, -15.319, -83.781, 50.693]
  Call Extruder(0.007)
  MoveL 3037 to (498.46, 491.94, 6.1) mm, rotated rx 0 ry 90 rz 0 deg; joints [-11.297, -26.989, 111.443, -15.286, -83.787, 50.688]
  Call Extruder(0.045)
  MoveL 3038 to (498.46, 490.4, 6.1) mm, rotated rx 0 ry 90 rz 0 deg; joints [-11.154, -26.994, 111.48, -15.142, -83.813, 50.667]
  Call Extruder(0.065)
  MoveL 3039 to (500.69, 490.4, 6.1) mm, rotated rx 0 ry 90 rz 0 deg; joints [-11.114, -26.956, 111.213, -15.108, -83.593, 50.722]
  Call Extruder(0.045)
  MoveL 3040 to (500.69, 491.94, 6.1) mm, rotated rx 0 ry 90 rz 0 deg; joints [-11.256, -26.95, 111.177, -15.251, -83.567, 50.744]
  Call Extruder(0.010)
  MoveL 3041 to (500.69, 492.29, 6.1) mm, rotated rx 0 ry 90 rz 0 deg; joints [-11.288, -26.949, 111.169, -15.284, -83.561, 50.749]
  Call Extruder(0.007)
  MoveL 3042 to (501.04, 492.29, 6.1) mm, rotated rx 0 ry 90 rz 0 deg; joints [-11.282, -26.943, 111.127, -15.279, -83.526, 50.758]
  Call Extruder(0.063)
  MoveL 3043 to (503.22, 492.29, 6.1) mm, rotated rx 0 ry 90 rz 0 deg; joints [-11.242, -26.904, 110.867, -15.245, -83.312, 50.813]
  Call Extruder(0.055)
  MoveL 3044 to (503.22, 490.4, 6.1) mm, rotated rx 0 ry 90 rz 0 deg; joints [-11.068, -26.911, 110.911, -15.069, -83.344, 50.785]
  Call Extruder(0.186)
  MoveL 3045 to (509.6, 490.4, 6.1) mm, rotated rx 0 ry 90 rz 0 deg; joints [-10.955, -26.792, 110.146, -14.976, -82.715, 50.942]
  Call Extruder(0.233)
  MoveL 3046 to (509.6, 498.4, 6.1) mm, rotated rx 0 ry 90 rz 0 deg; joints [-11.68, -26.761, 109.953, -15.712, -82.581, 51.068]
  Call Extruder(0.057)
  MoveL 3047 to (507.66, 498.4, 6.1) mm, rotated rx 0 ry 90 rz 0 deg; joints [-11.716, -26.798, 110.186, -15.742, -82.771, 51.018]
  Set speed (120.0 mm/s)
  MoveL 3048 to (507.66, 498.8, 6.1) mm, rotated rx 0 ry 90 rz 0 deg; joints [-11.753, -26.797, 110.176, -15.779, -82.764, 51.025]
  Set speed (1000.0 mm/s)
  MoveL 3049 to (506.96, 498.8, 6.1) mm, rotated rx 0 ry 90 rz 0 deg; joints [-11.766, -26.81, 110.26, -15.79, -82.833, 51.007]
  Set speed (1000.0 mm/s)
  MoveL 3050 to (490.68, 490.68, 6.1) mm, rotated rx 0 ry 90 rz 0 deg; joints [-11.324, -27.122, 112.395, -15.291, -84.577, 50.474]
  Set speed (1000.0 mm/s)
  MoveL 3051 to (490.68, 490.68, 6.2) mm, rotated rx 0 ry 90 rz 0 deg; joints [-11.324, -27.133, 112.4, -15.291, -84.572, 50.475]
  Set speed (30.0 mm/s)
  Call Extruder(0.767)
  MoveL 3052 to (509.32, 509.32, 6.2) mm, rotated rx 0 ry 90 rz 0 deg; joints [-12.669, -26.731, 109.708, -16.716, -82.409, 51.244]
  MoveL 3053 to (509.44, 509.44, 6.2) mm, rotated rx 0 ry 90 rz 0 deg; joints [-12.677, -26.728, 109.69, -16.726, -82.395, 51.249]
  Set speed (120.0 mm/s)
  MoveL 3054 to (508.74, 501.16, 6.2) mm, rotated rx 0 ry 90 rz 0 deg; joints [-11.946, -26.777, 109.993, -15.979, -82.613, 51.092]
  Set speed (30.0 mm/s)
  Call Extruder(0.336)
  MoveL 3055 to (500.58, 509.32, 6.2) mm, rotated rx 0 ry 90 rz 0 deg; joints [-12.847, -26.896, 110.754, -16.865, -83.257, 51.007]
  Set speed (120.0 mm/s)
  MoveL 3056 to (499.42, 509.32, 6.2) mm, rotated rx 0 ry 90 rz 0 deg; joints [-12.872, -26.917, 110.892, -16.885, -83.37, 50.975]
  Set speed (30.0 mm/s)
  Call Extruder(0.360)
  MoveL 3057 to (490.68, 500.58, 6.2) mm, rotated rx 0 ry 90 rz 0 deg; joints [-12.247, -27.1, 112.156, -16.224, -84.391, 50.608]
  Set speed (120.0 mm/s)
  MoveL 3058 to (490.68, 499.42, 6.2) mm, rotated rx 0 ry 90 rz 0 deg; joints [-12.139, -27.104, 112.186, -16.115, -84.412, 50.592]
  Set speed (30.0 mm/s)
  Call Extruder(0.282)
  MoveL 3059 to (497.53, 492.57, 6.2) mm, rotated rx 0 ry 90 rz 0 deg; joints [-11.372, -27.014, 111.544, -15.36, -83.863, 50.675]
  MoveL 3060 to (497.65, 492.45, 6.2) mm, rotated rx 0 ry 90 rz 0 deg; joints [-11.359, -27.012, 111.533, -15.346, -83.853, 50.676]
  Set speed (120.0 mm/s)
  MoveL 3061 to (498.8, 491.3, 6.2) mm, rotated rx 0 ry 90 rz 0 deg; joints [-11.232, -26.996, 111.423, -15.221, -83.759, 50.689]
  Set speed (30.0 mm/s)
  Call Extruder(0.026)
  MoveL 3062 to (499.42, 490.68, 6.2) mm, rotated rx 0 ry 90 rz 0 deg; joints [-11.163, -26.987, 111.364, -15.153, -83.709, 50.696]
  Set speed (120.0 mm/s)
  MoveL 3063 to (500.6, 492.32, 6.2) mm, rotated rx 0 ry 90 rz 0 deg; joints [-11.292, -26.961, 111.184, -15.288, -83.564, 50.749]
  Set speed (1000.0 mm/s)
  MoveL 3064 to (502.47, 492.57, 6.2) mm, rotated rx 0 ry 90 rz 0 deg; joints [-11.281, -26.927, 110.955, -15.283, -83.375, 50.8]
  Set speed (30.0 mm/s)
  Call Extruder(0.228)
  MoveL 3065 to (508.02, 498.12, 6.2) mm, rotated rx 0 ry 90 rz 0 deg; joints [-11.684, -26.803, 110.155, -15.711, -82.736, 51.025]
  MoveL 3066 to (508.14, 498.25, 6.2) mm, rotated rx 0 ry 90 rz 0 deg; joints [-11.693, -26.8, 110.137, -15.72, -82.721, 51.03]
  Set speed (120.0 mm/s)
  MoveL 3067 to (509.32, 490.68, 6.2) mm, rotated rx 0 ry 90 rz 0 deg; joints [-10.985, -26.807, 110.178, -15.006, -82.733, 50.941]
  Set speed (30.0 mm/s)
  Call Extruder(0.767)
  MoveL 3068 to (490.68, 509.32, 6.2) mm, rotated rx 0 ry 90 rz 0 deg; joints [-13.056, -27.068, 111.925, -17.042, -84.22, 50.733]
  MoveL 3069 to (490.56, 509.44, 6.2) mm, rotated rx 0 ry 90 rz 0 deg; joints [-13.07, -27.069, 111.937, -17.056, -84.23, 50.732]
  Set speed (120.0 mm/s)
  MoveL 3070 to (507.59, 498.33, 6.2) mm, rotated rx 0 ry 90 rz 0 deg; joints [-11.711, -26.81, 110.201, -15.737, -82.774, 51.017]
  Set speed (1000.0 mm/s)
  MoveL 3071 to (507.66, 498.4, 6.2) mm, rotated rx 0 ry 90 rz 0 deg; joints [-11.716, -26.809, 110.191, -15.742, -82.766, 51.02]
  Set speed (15.0 mm/s)
  Call Extruder(0.072)
  MoveL 3072 to (507.66, 500.88, 6.2) mm, rotated rx 0 ry 90 rz 0 deg; joints [-11.941, -26.799, 110.129, -15.97, -82.723, 51.06]
  Call Extruder(0.056)
  MoveL 3073 to (509.6, 500.88, 6.2) mm, rotated rx 0 ry 90 rz 0 deg; joints [-11.904, -26.762, 109.896, -15.94, -82.533, 51.11]
  Call Extruder(0.254)
  MoveL 3074 to (509.6, 509.6, 6.2) mm, rotated rx 0 ry 90 rz 0 deg; joints [-12.688, -26.724, 109.667, -16.738, -82.376, 51.256]
  Call Extruder(0.559)
  MoveL 3075 to (490.4, 509.6, 6.2) mm, rotated rx 0 ry 90 rz 0 deg; joints [-13.088, -27.071, 111.951, -17.074, -84.242, 50.73]
  MoveL 3076 to (490.4, 490.4, 6.2) mm, rotated rx 0 ry 90 rz 0 deg; joints [-11.303, -27.138, 112.44, -15.27, -84.605, 50.464]
  Call Extruder(0.163)
  MoveL 3077 to (496.01, 490.4, 6.2) mm, rotated rx 0 ry 90 rz 0 deg; joints [-11.199, -27.047, 111.776, -15.18, -84.05, 50.607]
  Call Extruder(0.055)
  MoveL 3078 to (496.01, 492.29, 6.2) mm, rotated rx 0 ry 90 rz 0 deg; joints [-11.375, -27.04, 111.731, -15.358, -84.017, 50.633]
  Call Extruder(0.063)
  MoveL 3079 to (498.17, 492.29, 6.2) mm, rotated rx 0 ry 90 rz 0 deg; joints [-11.335, -27.004, 111.475, -15.323, -83.804, 50.687]
  Call Extruder(0.010)
  MoveL 3080 to (498.52, 492.29, 6.2) mm, rotated rx 0 ry 90 rz 0 deg; joints [-11.328, -26.997, 111.433, -15.318, -83.77, 50.696]
  Call Extruder(0.007)
  MoveL 3081 to (498.52, 491.94, 6.2) mm, rotated rx 0 ry 90 rz 0 deg; joints [-11.296, -26.999, 111.441, -15.285, -83.776, 50.691]
  Call Extruder(0.045)
  MoveL 3082 to (498.52, 490.4, 6.2) mm, rotated rx 0 ry 90 rz 0 deg; joints [-11.153, -27.004, 111.478, -15.141, -83.802, 50.669]
  Call Extruder(0.062)
  MoveL 3083 to (500.63, 490.4, 6.2) mm, rotated rx 0 ry 90 rz 0 deg; joints [-11.115, -26.967, 111.226, -15.109, -83.594, 50.722]
  Call Extruder(0.045)
  MoveL 3084 to (500.63, 491.94, 6.2) mm, rotated rx 0 ry 90 rz 0 deg; joints [-11.257, -26.962, 111.19, -15.253, -83.568, 50.744]
  Call Extruder(0.010)
  MoveL 3085 to (500.63, 492.29, 6.2) mm, rotated rx 0 ry 90 rz 0 deg; joints [-11.289, -26.961, 111.181, -15.285, -83.562, 50.749]
  Call Extruder(0.007)
  MoveL 3086 to (500.98, 492.29, 6.2) mm, rotated rx 0 ry 90 rz 0 deg; joints [-11.283, -26.954, 111.14, -15.28, -83.527, 50.758]
  Call Extruder(0.063)
  MoveL 3087 to (503.15, 492.29, 6.2) mm, rotated rx 0 ry 90 rz 0 deg; joints [-11.243, -26.916, 110.88, -15.247, -83.313, 50.813]
  Call Extruder(0.055)
  MoveL 3088 to (503.15, 490.4, 6.2) mm, rotated rx 0 ry 90 rz 0 deg; joints [-11.069, -26.922, 110.924, -15.071, -83.345, 50.785]
  Call Extruder(0.188)
  MoveL 3089 to (509.6, 490.4, 6.2) mm, rotated rx 0 ry 90 rz 0 deg; joints [-10.955, -26.802, 110.151, -14.976, -82.71, 50.943]
  Call Extruder(0.233)
  MoveL 3090 to (509.6, 498.4, 6.2) mm, rotated rx 0 ry 90 rz 0 deg; joints [-11.68, -26.772, 109.958, -15.712, -82.576, 51.069]
  Call Extruder(0.056)
  MoveL 3091 to (507.66, 498.4, 6.2) mm, rotated rx 0 ry 90 rz 0 deg; joints [-11.716, -26.809, 110.191, -15.742, -82.766, 51.02]
  Set speed (120.0 mm/s)
  MoveL 3092 to (507.66, 498.8, 6.2) mm, rotated rx 0 ry 90 rz 0 deg; joints [-11.753, -26.807, 110.181, -15.779, -82.759, 51.026]
  Set speed (1000.0 mm/s)
  MoveL 3093 to (506.96, 498.8, 6.2) mm, rotated rx 0 ry 90 rz 0 deg; joints [-11.766, -26.821, 110.265, -15.79, -82.828, 51.008]
  Set speed (1000.0 mm/s)
  MoveL 3094 to (490.68, 490.68, 6.2) mm, rotated rx 0 ry 90 rz 0 deg; joints [-11.324, -27.133, 112.4, -15.291, -84.572, 50.475]
  Set speed (1000.0 mm/s)
  MoveL 3095 to (490.68, 490.68, 6.3) mm, rotated rx 0 ry 90 rz 0 deg; joints [-11.324, -27.143, 112.405, -15.292, -84.567, 50.476]
  Set speed (30.0 mm/s)
  Call Extruder(0.767)
  MoveL 3096 to (509.32, 509.32, 6.3) mm, rotated rx 0 ry 90 rz 0 deg; joints [-12.669, -26.742, 109.714, -16.717, -82.404, 51.245]
  MoveL 3097 to (509.44, 509.44, 6.3) mm, rotated rx 0 ry 90 rz 0 deg; joints [-12.677, -26.739, 109.696, -16.726, -82.39, 51.25]
  Set speed (120.0 mm/s)
  MoveL 3098 to (508.74, 501.16, 6.3) mm, rotated rx 0 ry 90 rz 0 deg; joints [-11.946, -26.788, 109.998, -15.979, -82.608, 51.093]
  Set speed (30.0 mm/s)
  Call Extruder(0.336)
  MoveL 3099 to (500.58, 509.32, 6.3) mm, rotated rx 0 ry 90 rz 0 deg; joints [-12.847, -26.907, 110.759, -16.865, -83.252, 51.009]
  Set speed (120.0 mm/s)
  MoveL 3100 to (499.42, 509.32, 6.3) mm, rotated rx 0 ry 90 rz 0 deg; joints [-12.872, -26.928, 110.897, -16.885, -83.365, 50.977]
  Set speed (30.0 mm/s)
  Call Extruder(0.360)
  MoveL 3101 to (490.68, 500.58, 6.3) mm, rotated rx 0 ry 90 rz 0 deg; joints [-12.247, -27.11, 112.162, -16.224, -84.385, 50.609]
  Set speed (120.0 mm/s)
  MoveL 3102 to (490.68, 499.42, 6.3) mm, rotated rx 0 ry 90 rz 0 deg; joints [-12.139, -27.114, 112.191, -16.115, -84.407, 50.593]
  Set speed (30.0 mm/s)
  Call Extruder(0.282)
  MoveL 3103 to (497.53, 492.57, 6.3) mm, rotated rx 0 ry 90 rz 0 deg; joints [-11.372, -27.024, 111.55, -15.36, -83.858, 50.676]
  MoveL 3104 to (497.65, 492.45, 6.3) mm, rotated rx 0 ry 90 rz 0 deg; joints [-11.359, -27.022, 111.538, -15.346, -83.848, 50.678]
  Set speed (120.0 mm/s)
  MoveL 3105 to (498.85, 491.24, 6.3) mm, rotated rx 0 ry 90 rz 0 deg; joints [-11.225, -27.006, 111.423, -15.215, -83.749, 50.691]
  Set speed (30.0 mm/s)
  Call Extruder(0.023)
  MoveL 3106 to (499.42, 490.68, 6.3) mm, rotated rx 0 ry 90 rz 0 deg; joints [-11.163, -26.998, 111.369, -15.153, -83.703, 50.697]
  Set speed (120.0 mm/s)
  MoveL 3107 to (500.54, 492.32, 6.3) mm, rotated rx 0 ry 90 rz 0 deg; joints [-11.293, -26.973, 111.197, -15.289, -83.565, 50.749]
  Set speed (1000.0 mm/s)
  MoveL 3108 to (502.47, 492.57, 6.3) mm, rotated rx 0 ry 90 rz 0 deg; joints [-11.281, -26.937, 110.96, -15.283, -83.37, 50.801]
  Set speed (30.0 mm/s)
  Call Extruder(0.228)
  MoveL 3109 to (508.02, 498.12, 6.3) mm, rotated rx 0 ry 90 rz 0 deg; joints [-11.684, -26.814, 110.16, -15.711, -82.731, 51.026]
  MoveL 3110 to (508.14, 498.24, 6.3) mm, rotated rx 0 ry 90 rz 0 deg; joints [-11.693, -26.811, 110.142, -15.72, -82.717, 51.031]
  Set speed (120.0 mm/s)
  MoveL 3111 to (509.32, 490.68, 6.3) mm, rotated rx 0 ry 90 rz 0 deg; joints [-10.985, -26.817, 110.183, -15.006, -82.728, 50.942]
  Set speed (30.0 mm/s)
  Call Extruder(0.767)
  MoveL 3112 to (490.68, 509.32, 6.3) mm, rotated rx 0 ry 90 rz 0 deg; joints [-13.056, -27.078, 111.931, -17.042, -84.215, 50.735]
  MoveL 3113 to (490.56, 509.44, 6.3) mm, rotated rx 0 ry 90 rz 0 deg; joints [-13.07, -27.08, 111.942, -17.056, -84.225, 50.733]
  Set speed (120.0 mm/s)
  MoveL 3114 to (507.59, 498.33, 6.3) mm, rotated rx 0 ry 90 rz 0 deg; joints [-11.711, -26.821, 110.207, -15.737, -82.769, 51.018]
  Set speed (1000.0 mm/s)
  MoveL 3115 to (507.66, 498.4, 6.3) mm, rotated rx 0 ry 90 rz 0 deg; joints [-11.716, -26.819, 110.197, -15.742, -82.761, 51.021]
  Set speed (15.0 mm/s)
  Call Extruder(0.072)
  MoveL 3116 to (507.66, 500.88, 6.3) mm, rotated rx 0 ry 90 rz 0 deg; joints [-11.941, -26.809, 110.134, -15.97, -82.718, 51.061]
  Call Extruder(0.056)
  MoveL 3117 to (509.6, 500.88, 6.3) mm, rotated rx 0 ry 90 rz 0 deg; joints [-11.904, -26.772, 109.901, -15.94, -82.528, 51.111]
  Call Extruder(0.254)
  MoveL 3118 to (509.6, 509.6, 6.3) mm, rotated rx 0 ry 90 rz 0 deg; joints [-12.688, -26.735, 109.672, -16.738, -82.371, 51.257]
  Call Extruder(0.559)
  MoveL 3119 to (490.4, 509.6, 6.3) mm, rotated rx 0 ry 90 rz 0 deg; joints [-13.088, -27.082, 111.956, -17.074, -84.237, 50.731]
  MoveL 3120 to (490.4, 490.4, 6.3) mm, rotated rx 0 ry 90 rz 0 deg; joints [-11.303, -27.149, 112.445, -15.27, -84.599, 50.466]
  Call Extruder(0.165)
  MoveL 3121 to (496.07, 490.4, 6.3) mm, rotated rx 0 ry 90 rz 0 deg; joints [-11.198, -27.056, 111.774, -15.179, -84.039, 50.609]
  Call Extruder(0.055)
  MoveL 3122 to (496.07, 492.29, 6.3) mm, rotated rx 0 ry 90 rz 0 deg; joints [-11.374, -27.05, 111.729, -15.357, -84.006, 50.635]
  Call Extruder(0.063)
  MoveL 3123 to (498.23, 492.29, 6.3) mm, rotated rx 0 ry 90 rz 0 deg; joints [-11.333, -27.013, 111.473, -15.323, -83.793, 50.69]
  Call Extruder(0.010)
  MoveL 3124 to (498.58, 492.29, 6.3) mm, rotated rx 0 ry 90 rz 0 deg; joints [-11.327, -27.007, 111.431, -15.317, -83.759, 50.699]
  Call Extruder(0.007)
  MoveL 3125 to (498.58, 491.94, 6.3) mm, rotated rx 0 ry 90 rz 0 deg; joints [-11.295, -27.008, 111.44, -15.284, -83.765, 50.694]
  Call Extruder(0.045)
  MoveL 3126 to (498.57, 490.4, 6.3) mm, rotated rx 0 ry 90 rz 0 deg; joints [-11.152, -27.014, 111.476, -15.14, -83.791, 50.672]
  Call Extruder(0.058)
  MoveL 3127 to (500.57, 490.4, 6.3) mm, rotated rx 0 ry 90 rz 0 deg; joints [-11.116, -26.979, 111.239, -15.11, -83.595, 50.722]
  Call Extruder(0.045)
  MoveL 3128 to (500.57, 491.94, 6.3) mm, rotated rx 0 ry 90 rz 0 deg; joints [-11.258, -26.973, 111.202, -15.254, -83.569, 50.744]
  Call Extruder(0.010)
  MoveL 3129 to (500.57, 492.29, 6.3) mm, rotated rx 0 ry 90 rz 0 deg; joints [-11.29, -26.972, 111.194, -15.286, -83.563, 50.749]
  Call Extruder(0.007)
  MoveL 3130 to (500.92, 492.29, 6.3) mm, rotated rx 0 ry 90 rz 0 deg; joints [-11.284, -26.966, 111.152, -15.281, -83.528, 50.758]
  Call Extruder(0.063)
  MoveL 3131 to (503.09, 492.29, 6.3) mm, rotated rx 0 ry 90 rz 0 deg; joints [-11.244, -26.927, 110.893, -15.248, -83.314, 50.812]
  Call Extruder(0.055)
  MoveL 3132 to (503.09, 490.4, 6.3) mm, rotated rx 0 ry 90 rz 0 deg; joints [-11.07, -26.934, 110.937, -15.072, -83.346, 50.785]
  Call Extruder(0.189)
  MoveL 3133 to (509.6, 490.4, 6.3) mm, rotated rx 0 ry 90 rz 0 deg; joints [-10.955, -26.813, 110.156, -14.976, -82.705, 50.945]
  Call Extruder(0.233)
  MoveL 3134 to (509.6, 498.4, 6.3) mm, rotated rx 0 ry 90 rz 0 deg; joints [-11.68, -26.782, 109.963, -15.712, -82.571, 51.071]
  Call Extruder(0.056)
  MoveL 3135 to (507.66, 498.4, 6.3) mm, rotated rx 0 ry 90 rz 0 deg; joints [-11.716, -26.819, 110.197, -15.742, -82.761, 51.021]
  Set speed (120.0 mm/s)
  MoveL 3136 to (507.66, 498.8, 6.3) mm, rotated rx 0 ry 90 rz 0 deg; joints [-11.752, -26.818, 110.187, -15.779, -82.754, 51.028]
  Set speed (1000.0 mm/s)
  MoveL 3137 to (506.96, 498.8, 6.3) mm, rotated rx 0 ry 90 rz 0 deg; joints [-11.766, -26.831, 110.271, -15.79, -82.823, 51.01]
  Set speed (1000.0 mm/s)
  MoveL 3138 to (490.68, 490.68, 6.3) mm, rotated rx 0 ry 90 rz 0 deg; joints [-11.324, -27.143, 112.405, -15.292, -84.567, 50.476]
  Set speed (1000.0 mm/s)
  MoveL 3139 to (490.68, 490.68, 6.4) mm, rotated rx 0 ry 90 rz 0 deg; joints [-11.324, -27.154, 112.411, -15.292, -84.562, 50.478]
  Set speed (30.0 mm/s)
  Call Extruder(0.767)
  MoveL 3140 to (509.32, 509.32, 6.4) mm, rotated rx 0 ry 90 rz 0 deg; joints [-12.669, -26.752, 109.719, -16.717, -82.399, 51.247]
  MoveL 3141 to (509.44, 509.44, 6.4) mm, rotated rx 0 ry 90 rz 0 deg; joints [-12.677, -26.749, 109.701, -16.726, -82.385, 51.252]
  Set speed (120.0 mm/s)
  MoveL 3142 to (508.74, 501.16, 6.4) mm, rotated rx 0 ry 90 rz 0 deg; joints [-11.945, -26.798, 110.003, -15.979, -82.603, 51.095]
  Set speed (30.0 mm/s)
  Call Extruder(0.336)
  MoveL 3143 to (500.58, 509.32, 6.4) mm, rotated rx 0 ry 90 rz 0 deg; joints [-12.847, -26.917, 110.764, -16.865, -83.247, 51.01]
  Set speed (120.0 mm/s)
  MoveL 3144 to (499.42, 509.32, 6.4) mm, rotated rx 0 ry 90 rz 0 deg; joints [-12.872, -26.938, 110.902, -16.885, -83.36, 50.978]
  Set speed (30.0 mm/s)
  Call Extruder(0.360)
  MoveL 3145 to (490.68, 500.58, 6.4) mm, rotated rx 0 ry 90 rz 0 deg; joints [-12.247, -27.121, 112.167, -16.224, -84.38, 50.611]
  Set speed (120.0 mm/s)
  MoveL 3146 to (490.68, 499.42, 6.4) mm, rotated rx 0 ry 90 rz 0 deg; joints [-12.139, -27.125, 112.197, -16.115, -84.402, 50.595]
  Set speed (30.0 mm/s)
  Call Extruder(0.282)
  MoveL 3147 to (497.53, 492.57, 6.4) mm, rotated rx 0 ry 90 rz 0 deg; joints [-11.372, -27.035, 111.555, -15.36, -83.852, 50.678]
  MoveL 3148 to (497.65, 492.45, 6.4) mm, rotated rx 0 ry 90 rz 0 deg; joints [-11.359, -27.033, 111.543, -15.347, -83.843, 50.679]
  Set speed (120.0 mm/s)
  MoveL 3149 to (498.91, 491.19, 6.4) mm, rotated rx 0 ry 90 rz 0 deg; joints [-11.218, -27.016, 111.423, -15.209, -83.739, 50.693]
  Set speed (30.0 mm/s)
  Call Extruder(0.021)
  MoveL 3150 to (499.42, 490.68, 6.4) mm, rotated rx 0 ry 90 rz 0 deg; joints [-11.163, -27.009, 111.374, -15.154, -83.698, 50.699]
  Set speed (120.0 mm/s)
  MoveL 3151 to (500.48, 492.32, 6.4) mm, rotated rx 0 ry 90 rz 0 deg; joints [-11.295, -26.984, 111.209, -15.29, -83.566, 50.749]
  Set speed (1000.0 mm/s)
  MoveL 3152 to (502.47, 492.58, 6.4) mm, rotated rx 0 ry 90 rz 0 deg; joints [-11.281, -26.948, 110.965, -15.283, -83.365, 50.803]
  Set speed (30.0 mm/s)
  Call Extruder(0.228)
  MoveL 3153 to (508.02, 498.12, 6.4) mm, rotated rx 0 ry 90 rz 0 deg; joints [-11.684, -26.824, 110.166, -15.711, -82.726, 51.027]
  MoveL 3154 to (508.14, 498.24, 6.4) mm, rotated rx 0 ry 90 rz 0 deg; joints [-11.693, -26.821, 110.148, -15.72, -82.712, 51.033]
  Set speed (120.0 mm/s)
  MoveL 3155 to (509.32, 490.68, 6.4) mm, rotated rx 0 ry 90 rz 0 deg; joints [-10.985, -26.828, 110.189, -15.006, -82.723, 50.944]
  Set speed (30.0 mm/s)
  Call Extruder(0.767)
  MoveL 3156 to (490.68, 509.32, 6.4) mm, rotated rx 0 ry 90 rz 0 deg; joints [-13.056, -27.089, 111.936, -17.043, -84.21, 50.737]
  MoveL 3157 to (490.56, 509.44, 6.4) mm, rotated rx 0 ry 90 rz 0 deg; joints [-13.07, -27.09, 111.947, -17.056, -84.219, 50.735]
  Set speed (120.0 mm/s)
  MoveL 3158 to (507.59, 498.33, 6.4) mm, rotated rx 0 ry 90 rz 0 deg; joints [-11.711, -26.831, 110.212, -15.737, -82.764, 51.02]
  Set speed (1000.0 mm/s)
  MoveL 3159 to (507.66, 498.4, 6.4) mm, rotated rx 0 ry 90 rz 0 deg; joints [-11.716, -26.83, 110.202, -15.742, -82.756, 51.023]
  Set speed (15.0 mm/s)
  Call Extruder(0.072)
  MoveL 3160 to (507.66, 500.88, 6.4) mm, rotated rx 0 ry 90 rz 0 deg; joints [-11.941, -26.82, 110.14, -15.97, -82.713, 51.062]
  Call Extruder(0.056)
